C07284=1060.234,-74.990,436.185,171.327,26.753,155.011
C07285=1060.227,-75.240,436.197,171.325,26.751,155.011
C07286=1060.222,-75.490,436.207,171.323,26.750,155.011
C07287=1060.215,-75.739,436.219,171.321,26.748,155.011
C07288=1060.208,-75.989,436.230,171.319,26.747,155.011
C07289=1060.202,-76.239,436.241,171.318,26.745,155.011
C07290=1060.196,-76.488,436.252,171.316,26.744,155.011
C07291=1060.190,-76.738,436.263,171.314,26.743,155.011
C07292=1060.184,-76.987,436.275,171.312,26.741,155.011
C07293=1060.178,-77.238,436.286,171.311,26.739,155.010
C07294=1060.172,-77.487,436.297,171.309,26.738,155.010
C07295=1060.166,-77.737,436.308,171.307,26.736,155.010
C07296=1060.159,-77.986,436.320,171.306,26.735,155.010
C07297=1060.154,-78.236,436.330,171.304,26.733,155.010
C07298=1060.147,-78.486,436.342,171.302,26.732,155.010
C07299=1060.142,-78.735,436.353,171.301,26.731,155.010
C07300=1060.135,-78.985,436.364,171.299,26.729,155.010
C07301=1060.130,-79.235,436.375,171.297,26.728,155.010
C07302=1060.123,-79.485,436.387,171.294,26.726,155.010
C07303=1060.117,-79.734,436.398,171.293,26.725,155.010
C07304=1060.111,-79.983,436.408,171.291,26.723,155.010
C07305=1060.104,-80.233,436.419,171.289,26.722,155.010
C07306=1060.099,-80.483,436.430,171.288,26.721,155.010
C07307=1060.092,-80.733,436.441,171.286,26.719,155.009
C07308=1060.086,-80.982,436.451,171.284,26.718,155.009
C07309=1060.079,-81.232,436.463,171.282,26.716,155.009
C07310=1060.074,-81.482,436.474,171.281,26.715,155.009
C07311=1060.067,-81.732,436.485,171.279,26.714,155.009
C07312=1060.061,-81.981,436.495,171.277,26.712,155.009
C07313=1060.054,-82.264,436.508,171.275,26.711,155.009
C07314=1060.047,-82.546,436.520,171.273,26.709,155.009
C07315=1060.039,-82.829,436.533,171.271,26.708,155.009
C07316=1060.033,-83.111,436.545,171.269,26.706,155.009
C07317=1060.026,-83.361,436.555,171.267,26.704,155.009
C07318=1060.021,-83.611,436.566,171.265,26.703,155.009
C07319=1060.014,-83.861,436.578,171.263,26.702,155.009
C07320=1060.008,-84.110,436.588,171.262,26.700,155.009
C07321=1060.002,-84.359,436.599,171.260,26.699,155.009
C07322=1059.996,-84.610,436.610,171.258,26.698,155.008
C07323=1059.990,-84.859,436.621,171.256,26.696,155.008
C07324=1059.983,-85.109,436.632,171.255,26.695,155.008
C07325=1059.977,-85.359,436.642,171.253,26.694,155.008
C07326=1059.971,-85.608,436.653,171.251,26.692,155.008
C07327=1059.964,-85.858,436.664,171.249,26.691,155.008
C07328=1059.959,-86.107,436.675,171.248,26.690,155.008
C07329=1059.953,-86.357,436.686,171.245,26.688,155.008
C07330=1059.946,-86.607,436.696,171.243,26.687,155.008
C07331=1059.940,-86.856,436.707,171.242,26.686,155.008
C07332=1059.934,-87.106,436.718,171.240,26.684,155.008
C07333=1059.927,-87.356,436.729,171.238,26.683,155.008
C07334=1059.921,-87.605,436.740,171.236,26.682,155.008
C07335=1059.915,-87.855,436.751,171.235,26.681,155.008
C07336=1059.909,-88.105,436.760,171.233,26.679,155.008
C07337=1059.903,-88.355,436.771,171.231,26.678,155.008
C07338=1059.897,-88.604,436.782,171.229,26.677,155.008
C07339=1059.890,-88.854,436.793,171.228,26.676,155.008
C07340=1059.885,-89.103,436.804,171.226,26.674,155.007
C07341=1059.879,-89.353,436.815,171.224,26.673,155.007
C07342=1059.872,-89.603,436.824,171.222,26.672,155.007
C07343=1059.866,-89.853,436.835,171.220,26.670,155.007
C07344=1059.861,-90.102,436.846,171.218,26.669,155.007
C07345=1059.854,-90.352,436.857,171.216,26.667,155.007
C07346=1059.848,-90.602,436.868,171.215,26.666,155.007
C07347=1059.841,-90.851,436.878,171.213,26.665,155.007
C07348=1059.836,-91.101,436.888,171.211,26.664,155.007
C07349=1059.830,-91.351,436.899,171.209,26.663,155.007
C07350=1059.823,-91.600,436.910,171.208,26.662,155.007
C07351=1059.817,-91.850,436.921,171.206,26.660,155.007
C07352=1059.812,-92.100,436.931,171.204,26.659,155.007
C07353=1059.805,-92.350,436.941,171.202,26.658,155.007
C07354=1059.799,-92.599,436.952,171.201,26.656,155.007
C07355=1059.793,-92.849,436.963,171.199,26.655,155.007
C07356=1059.787,-93.099,436.973,171.197,26.654,155.007
C07357=1059.781,-93.349,436.984,171.194,26.653,155.007
C07358=1059.774,-93.598,436.994,171.193,26.651,155.007
C07359=1059.769,-93.848,437.004,171.191,26.650,155.007
C07360=1059.762,-94.097,437.015,171.189,26.649,155.007
C07361=1059.757,-94.347,437.026,171.187,26.648,155.007
C07362=1059.750,-94.597,437.037,171.186,26.646,155.007
C07363=1059.744,-94.847,437.046,171.184,26.645,155.007
C07364=1059.738,-95.096,437.057,171.182,26.644,155.007
C07365=1059.732,-95.346,437.067,171.180,26.643,155.007
C07366=1059.727,-95.596,437.078,171.179,26.642,155.007
C07367=1059.719,-95.846,437.088,171.177,26.641,155.007
C07368=1059.714,-96.096,437.099,171.175,26.639,155.006
C07369=1059.708,-96.345,437.109,171.173,26.638,155.006
C07370=1059.702,-96.594,437.120,171.172,26.637,155.006
C07371=1059.696,-96.844,437.130,171.169,26.635,155.006
C07372=1059.690,-97.094,437.140,171.167,26.634,155.006
C07373=1059.684,-97.344,437.150,171.165,26.633,155.006
C07374=1059.677,-97.594,437.161,171.164,26.632,155.006
C07375=1059.672,-97.843,437.172,171.162,26.631,155.006
C07376=1059.666,-98.093,437.181,171.160,26.629,155.006
C07377=1059.659,-98.377,437.193,171.158,26.628,155.006
C07378=1059.651,-98.662,437.205,171.156,26.627,155.006
C07379=1059.644,-98.947,437.217,171.154,26.626,155.006
C07380=1059.637,-99.232,437.229,171.152,26.625,155.006
C07381=1059.631,-99.482,437.238,171.150,26.623,155.006
C07382=1059.625,-99.731,437.249,171.148,26.623,155.006
C07383=1059.619,-99.981,437.259,171.146,26.622,155.006
C07384=1059.612,-100.231,437.270,171.144,26.620,155.006
C07385=1059.606,-100.481,437.279,171.142,26.619,155.006
C07386=1059.600,-100.730,437.290,171.140,26.618,155.006
C07387=1059.594,-100.980,437.300,171.139,26.617,155.006
C07388=1059.588,-101.230,437.309,171.137,26.616,155.006
C07389=1059.582,-101.479,437.320,171.135,26.615,155.006
C07390=1059.576,-101.729,437.330,171.133,26.614,155.006
C07391=1059.569,-101.979,437.340,171.132,26.613,155.006
C07392=1059.563,-102.229,437.350,171.130,26.612,155.006
C07393=1059.557,-102.478,437.361,171.128,26.611,155.006
C07394=1059.551,-102.728,437.370,171.126,26.610,155.006
C07395=1059.545,-102.977,437.381,171.123,26.609,155.006
C07396=1059.539,-103.227,437.391,171.122,26.608,155.006
C07397=1059.533,-103.477,437.400,171.120,26.606,155.006
C07398=1059.527,-103.726,437.411,171.118,26.606,155.007
C07399=1059.521,-103.976,437.421,171.116,26.605,155.006
C07400=1059.515,-104.226,437.430,171.114,26.604,155.006
C07401=1059.508,-104.476,437.442,171.113,26.602,155.006
C07402=1059.502,-104.726,437.451,171.111,26.602,155.007
C07403=1059.496,-104.975,437.461,171.109,26.601,155.007
C07404=1059.489,-105.225,437.471,171.107,26.600,155.007
C07405=1059.484,-105.475,437.481,171.106,26.598,155.006
C07406=1059.478,-105.724,437.491,171.104,26.598,155.007
C07407=1059.471,-105.974,437.501,171.102,26.597,155.007
C07408=1059.465,-106.224,437.511,171.099,26.595,155.007
C07409=1059.459,-106.473,437.521,171.097,26.595,155.007
C07410=1059.453,-106.723,437.531,171.096,26.594,155.007
C07411=1059.447,-106.973,437.541,171.094,26.592,155.007
C07412=1059.441,-107.223,437.550,171.092,26.592,155.007
C07413=1059.435,-107.472,437.561,171.090,26.591,155.007
C07414=1059.429,-107.722,437.571,171.088,26.590,155.007
C07415=1059.423,-107.972,437.580,171.087,26.589,155.007
C07416=1059.417,-108.222,437.590,171.085,26.588,155.007
C07417=1059.410,-108.472,437.600,171.083,26.587,155.007
C07418=1059.403,-108.721,437.610,171.081,26.586,155.007
C07419=1059.397,-108.971,437.619,171.079,26.585,155.007
C07420=1059.392,-109.221,437.630,171.077,26.584,155.007
C07421=1059.385,-109.470,437.640,171.075,26.583,155.007
C07422=1059.379,-109.720,437.649,171.073,26.583,155.007
C07423=1059.373,-109.970,437.659,171.071,26.581,155.007
C07424=1059.367,-110.220,437.669,171.069,26.581,155.007
C07425=1059.361,-110.470,437.678,171.068,26.580,155.007
C07426=1059.354,-110.719,437.688,171.066,26.579,155.007
C07427=1059.348,-110.969,437.698,171.064,26.578,155.007
C07428=1059.342,-111.218,437.708,171.062,26.577,155.007
C07429=1059.336,-111.469,437.718,171.060,26.576,155.007
C07430=1059.330,-111.718,437.727,171.058,26.576,155.007
C07431=1059.324,-111.968,437.737,171.057,26.575,155.007
C07432=1059.318,-112.218,437.746,171.055,26.574,155.007
C07433=1059.311,-112.467,437.757,171.053,26.573,155.007
C07434=1059.305,-112.717,437.766,171.050,26.572,155.008
C07435=1059.299,-112.967,437.776,171.048,26.571,155.008
C07436=1059.293,-113.217,437.785,171.047,26.570,155.008
C07437=1059.287,-113.466,437.795,171.045,26.569,155.008
C07438=1059.281,-113.716,437.805,171.043,26.569,155.008
C07439=1059.275,-113.965,437.814,171.041,26.567,155.008
C07440=1059.269,-114.215,437.823,171.039,26.567,155.008
C07441=1059.262,-114.499,437.834,171.037,26.566,155.008
C07442=1059.255,-114.782,437.846,171.035,26.565,155.008
C07443=1059.248,-115.065,437.857,171.033,26.564,155.008
C07444=1059.241,-115.348,437.867,171.031,26.563,155.008
C07445=1059.235,-115.598,437.877,171.029,26.563,155.008
C07446=1059.229,-115.847,437.886,171.026,26.561,155.008
C07447=1059.222,-116.097,437.896,171.025,26.561,155.008
C07448=1059.216,-116.347,437.905,171.023,26.560,155.008
C07449=1059.210,-116.597,437.915,171.021,26.559,155.008
C07450=1059.204,-116.847,437.924,171.019,26.558,155.008
C07451=1059.198,-117.096,437.934,171.017,26.558,155.009
C07452=1059.192,-117.346,437.944,171.015,26.557,155.008
C07453=1059.185,-117.596,437.953,171.014,26.556,155.009
C07454=1059.179,-117.846,437.963,171.012,26.556,155.009
C07455=1059.174,-118.095,437.972,171.010,26.555,155.009
C07456=1059.167,-118.345,437.981,171.008,26.554,155.009
C07457=1059.161,-118.594,437.991,171.006,26.553,155.009
C07458=1059.155,-118.844,438.001,171.004,26.553,155.009
C07459=1059.148,-119.094,438.010,171.001,26.552,155.009
C07460=1059.142,-119.344,438.019,171.000,26.551,155.009
C07461=1059.136,-119.593,438.029,170.998,26.550,155.009
C07462=1059.130,-119.844,438.038,170.996,26.550,155.009
C07463=1059.124,-120.094,438.047,170.994,26.549,155.009
C07464=1059.118,-120.343,438.056,170.992,26.548,155.009
C07465=1059.112,-120.592,438.066,170.990,26.547,155.009
C07466=1059.106,-120.842,438.075,170.989,26.547,155.010
C07467=1059.100,-121.092,438.085,170.987,26.546,155.010
C07468=1059.093,-121.342,438.094,170.985,26.546,155.010
C07469=1059.087,-121.592,438.103,170.983,26.545,155.010
C07470=1059.081,-121.842,438.112,170.981,26.544,155.010
C07471=1059.075,-122.091,438.122,170.979,26.544,155.010
C07472=1059.069,-122.341,438.131,170.976,26.543,155.010
C07473=1059.063,-122.590,438.141,170.975,26.542,155.010
C07474=1059.057,-122.840,438.150,170.973,26.542,155.010
C07475=1059.050,-123.090,438.159,170.971,26.541,155.010
C07476=1059.044,-123.340,438.168,170.969,26.540,155.010
C07477=1059.038,-123.589,438.177,170.967,26.539,155.010
C07478=1059.032,-123.839,438.187,170.965,26.539,155.011
C07479=1059.026,-124.089,438.196,170.963,26.538,155.011
C07480=1059.020,-124.339,438.205,170.962,26.538,155.011
C07481=1059.013,-124.589,438.214,170.960,26.537,155.011
C07482=1059.008,-124.838,438.223,170.958,26.537,155.011
C07483=1059.002,-125.088,438.232,170.956,26.536,155.011
C07484=1058.996,-125.338,438.242,170.954,26.536,155.011
C07485=1058.989,-125.588,438.251,170.952,26.535,155.011
C07486=1058.983,-125.837,438.260,170.949,26.534,155.011
C07487=1058.977,-126.088,438.269,170.948,26.534,155.011
C07488=1058.970,-126.337,438.278,170.946,26.533,155.012
C07489=1058.964,-126.586,438.287,170.944,26.532,155.012
C07490=1058.958,-126.837,438.296,170.942,26.532,155.012
C07491=1058.952,-127.087,438.306,170.940,26.531,155.012
C07492=1058.946,-127.335,438.314,170.938,26.531,155.012
C07493=1058.940,-127.586,438.323,170.936,26.530,155.012
C07494=1058.934,-127.836,438.333,170.934,26.530,155.012
C07495=1058.929,-128.085,438.343,170.933,26.529,155.012
C07496=1058.925,-128.335,438.352,170.931,26.527,155.012
C07497=1058.923,-128.586,438.364,170.929,26.525,155.012
C07498=1058.921,-128.837,438.375,170.928,26.522,155.012
C07499=1058.922,-129.087,438.388,170.927,26.519,155.011
C07500=1058.923,-129.337,438.401,170.926,26.515,155.011
C07501=1058.926,-129.589,438.415,170.925,26.511,155.010
C07502=1058.931,-129.840,438.429,170.924,26.505,155.009
C07503=1058.937,-130.091,438.445,170.924,26.500,155.008
C07504=1058.944,-130.341,438.461,170.923,26.494,155.007
C07505=1058.567,-130.364,438.262,170.876,26.654,155.040
C07506=1058.559,-130.114,438.246,170.876,26.661,155.041
C07507=1058.554,-129.864,438.232,170.877,26.666,155.042
C07508=1058.550,-129.612,438.217,170.878,26.671,155.043
C07509=1058.547,-129.361,438.203,170.878,26.676,155.044
C07510=1058.544,-129.110,438.189,170.879,26.680,155.044
C07511=1058.545,-128.860,438.177,170.880,26.683,155.045
C07512=1058.545,-128.609,438.165,170.882,26.686,155.045
C07513=1058.547,-128.358,438.154,170.883,26.688,155.045
C07514=1058.551,-128.109,438.144,170.884,26.690,155.045
C07515=1058.556,-127.859,438.135,170.886,26.691,155.046
C07516=1058.562,-127.609,438.125,170.889,26.692,155.045
C07517=1058.568,-127.359,438.115,170.891,26.692,155.045
C07518=1058.574,-127.109,438.107,170.893,26.692,155.045
C07519=1058.581,-126.860,438.098,170.894,26.693,155.045
C07520=1058.587,-126.610,438.088,170.896,26.693,155.045
C07521=1058.593,-126.360,438.080,170.898,26.694,155.045
C07522=1058.599,-126.110,438.071,170.900,26.694,155.045
C07523=1058.606,-125.860,438.061,170.902,26.695,155.045
C07524=1058.611,-125.611,438.052,170.904,26.695,155.044
C07525=1058.617,-125.361,438.043,170.906,26.696,155.044
C07526=1058.624,-125.111,438.034,170.908,26.696,155.044
C07527=1058.630,-124.861,438.024,170.910,26.697,155.044
C07528=1058.636,-124.611,438.016,170.912,26.698,155.044
C07529=1058.642,-124.361,438.006,170.914,26.698,155.044
C07530=1058.648,-124.112,437.997,170.916,26.699,155.044
C07531=1058.655,-123.863,437.988,170.918,26.700,155.044
C07532=1058.661,-123.613,437.978,170.920,26.701,155.044
C07533=1058.667,-123.362,437.969,170.922,26.701,155.044
C07534=1058.673,-123.113,437.960,170.924,26.702,155.044
C07535=1058.678,-122.864,437.951,170.925,26.702,155.043
C07536=1058.685,-122.614,437.942,170.927,26.703,155.043
C07537=1058.691,-122.364,437.933,170.929,26.703,155.043
C07538=1058.697,-122.114,437.923,170.931,26.704,155.043
C07539=1058.704,-121.864,437.914,170.933,26.705,155.043
C07540=1058.710,-121.614,437.904,170.935,26.705,155.043
C07541=1058.715,-121.365,437.895,170.937,26.706,155.043
C07542=1058.721,-121.115,437.885,170.939,26.707,155.043
C07543=1058.728,-120.866,437.876,170.941,26.707,155.043
C07544=1058.734,-120.615,437.868,170.943,26.708,155.043
C07545=1058.740,-120.366,437.858,170.945,26.709,155.043
C07546=1058.747,-120.116,437.848,170.947,26.710,155.043
C07547=1058.753,-119.866,437.839,170.949,26.710,155.042
C07548=1058.759,-119.616,437.829,170.951,26.711,155.042
C07549=1058.764,-119.367,437.820,170.952,26.712,155.042
C07550=1058.771,-119.117,437.811,170.954,26.712,155.042
C07551=1058.777,-118.868,437.801,170.956,26.713,155.042
C07552=1058.783,-118.618,437.791,170.958,26.713,155.042
C07553=1058.790,-118.368,437.782,170.961,26.715,155.042
C07554=1058.796,-118.118,437.774,170.963,26.715,155.042
C07555=1058.802,-117.868,437.764,170.964,26.716,155.042
C07556=1058.808,-117.618,437.754,170.966,26.716,155.042
C07557=1058.814,-117.368,437.745,170.968,26.718,155.042
C07558=1058.820,-117.119,437.735,170.970,26.718,155.042
C07559=1058.826,-116.870,437.726,170.972,26.719,155.042
C07560=1058.832,-116.620,437.717,170.974,26.720,155.042
C07561=1058.838,-116.370,437.707,170.975,26.720,155.042
C07562=1058.845,-116.120,437.697,170.977,26.721,155.041
C07563=1058.851,-115.870,437.688,170.979,26.722,155.041
C07564=1058.857,-115.621,437.678,170.981,26.723,155.041
C07565=1058.863,-115.371,437.669,170.984,26.723,155.041
C07566=1058.870,-115.087,437.658,170.986,26.725,155.041
C07567=1058.878,-114.804,437.647,170.987,26.725,155.041
C07568=1058.884,-114.522,437.636,170.990,26.726,155.041
C07569=1058.891,-114.238,437.625,170.992,26.727,155.041
C07570=1058.897,-113.988,437.615,170.994,26.728,155.041
C07571=1058.903,-113.738,437.606,170.996,26.729,155.041
C07572=1058.910,-113.489,437.596,170.998,26.729,155.041
C07573=1058.916,-113.239,437.587,170.999,26.730,155.041
C07574=1058.922,-112.989,437.577,171.001,26.731,155.041
C07575=1058.928,-112.740,437.567,171.003,26.732,155.041
C07576=1058.934,-112.490,437.557,171.006,26.733,155.041
C07577=1058.941,-112.240,437.548,171.008,26.734,155.041
C07578=1058.946,-111.990,437.538,171.009,26.735,155.041
C07579=1058.952,-111.740,437.528,171.011,26.735,155.040
C07580=1058.958,-111.490,437.519,171.013,26.736,155.041
C07581=1058.965,-111.241,437.509,171.015,26.737,155.040
C07582=1058.971,-110.992,437.499,171.017,26.738,155.040
C07583=1058.977,-110.742,437.489,171.019,26.739,155.040
C07584=1058.983,-110.492,437.480,171.020,26.740,155.040
C07585=1058.990,-110.242,437.470,171.022,26.741,155.040
C07586=1058.996,-109.992,437.460,171.024,26.741,155.040
C07587=1059.002,-109.743,437.451,171.026,26.743,155.040
C07588=1059.008,-109.493,437.440,171.029,26.743,155.040
C07589=1059.014,-109.243,437.430,171.030,26.744,155.040
C07590=1059.020,-108.993,437.421,171.032,26.745,155.040
C07591=1059.026,-108.744,437.411,171.034,26.746,155.040
C07592=1059.033,-108.494,437.401,171.036,26.747,155.040
C07593=1059.039,-108.245,437.391,171.038,26.748,155.040
C07594=1059.045,-107.995,437.382,171.040,26.748,155.040
C07595=1059.051,-107.745,437.372,171.041,26.750,155.040
C07596=1059.057,-107.496,437.361,171.043,26.751,155.040
C07597=1059.063,-107.246,437.352,171.045,26.751,155.040
C07598=1059.069,-106.996,437.342,171.047,26.752,155.040
C07599=1059.075,-106.746,437.333,171.049,26.753,155.040
C07600=1059.082,-106.496,437.321,171.051,26.754,155.040
C07601=1059.088,-106.246,437.312,171.053,26.755,155.040
C07602=1059.094,-105.996,437.302,171.055,26.757,155.040
C07603=1059.101,-105.747,437.292,171.057,26.757,155.040
C07604=1059.106,-105.497,437.282,171.059,26.758,155.040
C07605=1059.112,-105.247,437.272,171.060,26.759,155.040
C07606=1059.119,-104.998,437.262,171.062,26.760,155.040
C07607=1059.125,-104.748,437.252,171.064,26.761,155.040
C07608=1059.130,-104.498,437.242,171.066,26.762,155.040
C07609=1059.137,-104.249,437.232,171.067,26.763,155.040
C07610=1059.143,-103.999,437.222,171.069,26.764,155.040
C07611=1059.148,-103.749,437.212,171.071,26.765,155.040
C07612=1059.155,-103.500,437.202,171.073,26.766,155.040
C07613=1059.162,-103.249,437.192,171.076,26.768,155.040
C07614=1059.168,-103.000,437.182,171.077,26.768,155.040
C07615=1059.174,-102.750,437.172,171.079,26.769,155.040
C07616=1059.180,-102.501,437.161,171.081,26.770,155.040
C07617=1059.186,-102.251,437.152,171.083,26.772,155.040
C07618=1059.192,-102.001,437.142,171.085,26.773,155.040
C07619=1059.198,-101.752,437.131,171.086,26.773,155.040
C07620=1059.204,-101.502,437.122,171.088,26.774,155.040
C07621=1059.210,-101.253,437.111,171.090,26.775,155.040
C07622=1059.217,-101.002,437.101,171.092,26.777,155.040
C07623=1059.223,-100.753,437.091,171.094,26.778,155.040
C07624=1059.229,-100.503,437.080,171.095,26.778,155.040
C07625=1059.235,-100.254,437.070,171.098,26.780,155.040
C07626=1059.241,-100.004,437.061,171.100,26.781,155.040
C07627=1059.247,-99.754,437.050,171.102,26.782,155.040
C07628=1059.254,-99.504,437.040,171.103,26.783,155.040
C07629=1059.260,-99.254,437.029,171.105,26.784,155.040
C07630=1059.267,-98.969,437.018,171.107,26.785,155.040
C07631=1059.273,-98.685,437.006,171.110,26.787,155.040
C07632=1059.281,-98.399,436.994,171.111,26.788,155.040
C07633=1059.288,-98.115,436.983,171.113,26.789,155.040
C07634=1059.294,-97.865,436.973,171.115,26.790,155.040
C07635=1059.300,-97.616,436.962,171.118,26.792,155.040
C07636=1059.307,-97.367,436.952,171.120,26.792,155.040
C07637=1059.313,-97.116,436.942,171.121,26.793,155.040
C07638=1059.318,-96.866,436.931,171.123,26.795,155.040
C07639=1059.325,-96.617,436.921,171.125,26.796,155.040
C07640=1059.330,-96.367,436.910,171.127,26.797,155.040
C07641=1059.337,-96.118,436.900,171.128,26.798,155.040
C07642=1059.342,-95.868,436.890,171.130,26.800,155.040
C07643=1059.349,-95.618,436.879,171.132,26.801,155.040
C07644=1059.355,-95.368,436.868,171.134,26.802,155.040
C07645=1059.361,-95.118,436.858,171.135,26.803,155.040
C07646=1059.367,-94.869,436.848,171.137,26.804,155.040
C07647=1059.373,-94.620,436.837,171.139,26.805,155.040
C07648=1059.379,-94.370,436.827,171.142,26.807,155.040
C07649=1059.385,-94.120,436.816,171.143,26.808,155.040
C07650=1059.391,-93.870,436.805,171.145,26.809,155.040
C07651=1059.397,-93.620,436.796,171.147,26.811,155.040
C07652=1059.403,-93.371,436.785,171.149,26.812,155.040
C07653=1059.410,-93.121,436.774,171.150,26.813,155.040
C07654=1059.415,-92.871,436.764,171.152,26.814,155.040
C07655=1059.421,-92.621,436.753,171.154,26.815,155.040
C07656=1059.428,-92.372,436.743,171.156,26.816,155.040
C07657=1059.433,-92.123,436.732,171.157,26.817,155.040
C07658=1059.440,-91.872,436.722,171.159,26.819,155.040
C07659=1059.446,-91.623,436.711,171.161,26.820,155.040
C07660=1059.452,-91.373,436.700,171.163,26.821,155.040
C07661=1059.459,-91.123,436.690,171.164,26.823,155.040
C07662=1059.464,-90.874,436.679,171.167,26.824,155.040
C07663=1059.470,-90.624,436.669,171.169,26.825,155.040
C07664=1059.476,-90.375,436.658,171.171,26.826,155.040
C07665=1059.483,-90.124,436.647,171.172,26.828,155.041
C07666=1059.489,-89.875,436.637,171.174,26.829,155.041
C07667=1059.495,-89.626,436.626,171.176,26.830,155.041
C07668=1059.501,-89.375,436.615,171.178,26.831,155.041
C07669=1059.507,-89.126,436.605,171.179,26.833,155.041
C07670=1059.513,-88.876,436.594,171.181,26.834,155.041
C07671=1059.519,-88.627,436.583,171.183,26.835,155.041
C07672=1059.526,-88.377,436.573,171.185,26.837,155.041
C07673=1059.532,-88.127,436.562,171.186,26.838,155.041
C07674=1059.537,-87.878,436.551,171.188,26.839,155.041
C07675=1059.544,-87.627,436.541,171.191,26.841,155.041
C07676=1059.550,-87.378,436.530,171.193,26.842,155.041
C07677=1059.556,-87.128,436.519,171.194,26.843,155.041
C07678=1059.563,-86.879,436.509,171.196,26.845,155.041
C07679=1059.569,-86.629,436.498,171.198,26.846,155.041
C07680=1059.574,-86.380,436.487,171.200,26.847,155.041
C07681=1059.581,-86.130,436.476,171.201,26.848,155.041
C07682=1059.587,-85.880,436.465,171.203,26.850,155.041
C07683=1059.593,-85.630,436.454,171.205,26.851,155.041
C07684=1059.600,-85.381,436.444,171.207,26.852,155.041
C07685=1059.606,-85.131,436.433,171.208,26.853,155.041
C07686=1059.612,-84.881,436.422,171.210,26.855,155.042
C07687=1059.618,-84.632,436.411,171.212,26.856,155.042
C07688=1059.625,-84.382,436.400,171.213,26.857,155.042
C07689=1059.631,-84.132,436.389,171.216,26.859,155.042
C07690=1059.636,-83.883,436.378,171.218,26.860,155.042
C07691=1059.643,-83.633,436.368,171.220,26.862,155.042
C07692=1059.649,-83.383,436.357,171.221,26.863,155.042
C07693=1059.655,-83.133,436.346,171.223,26.864,155.042
C07694=1059.662,-82.851,436.334,171.225,26.866,155.042
C07695=1059.669,-82.569,436.322,171.227,26.868,155.042
C07696=1059.676,-82.286,436.309,171.229,26.869,155.042
C07697=1059.684,-82.004,436.296,171.231,26.870,155.042
C07698=1059.689,-81.754,436.286,171.233,26.872,155.042
C07699=1059.696,-81.504,436.274,171.234,26.873,155.042
C07700=1059.702,-81.255,436.264,171.236,26.874,155.042
C07701=1059.709,-81.004,436.253,171.239,26.876,155.042
C07702=1059.714,-80.755,436.242,171.240,26.878,155.043
C07703=1059.721,-80.505,436.231,171.242,26.879,155.043
C07704=1059.727,-80.256,436.220,171.244,26.880,155.043
C07705=1059.733,-80.005,436.209,171.246,26.882,155.043
C07706=1059.739,-79.756,436.198,171.247,26.883,155.043
C07707=1059.746,-79.506,436.187,171.249,26.884,155.043
C07708=1059.752,-79.257,436.175,171.251,26.885,155.043
C07709=1059.758,-79.007,436.164,171.253,26.887,155.043
C07710=1059.764,-78.758,436.154,171.254,26.888,155.043
C07711=1059.770,-78.508,436.143,171.256,26.890,155.043
C07712=1059.777,-78.258,436.132,171.258,26.892,155.043
C07713=1059.783,-78.009,436.120,171.259,26.893,155.043
C07714=1059.789,-77.759,436.109,171.261,26.895,155.044
C07715=1059.795,-77.509,436.098,171.263,26.896,155.044
C07716=1059.801,-77.259,436.087,171.265,26.898,155.044
C07717=1059.807,-77.010,436.076,171.267,26.899,155.044
C07718=1059.813,-76.760,436.064,171.269,26.901,155.044
C07719=1059.819,-76.511,436.053,171.271,26.902,155.044
C07720=1059.825,-76.260,436.042,171.272,26.903,155.044
C07721=1059.831,-76.011,436.031,171.274,26.905,155.044
C07722=1059.838,-75.761,436.019,171.276,26.906,155.044
C07723=1059.844,-75.512,436.008,171.277,26.908,155.044
C07724=1059.850,-75.262,435.997,171.279,26.909,155.044
C07725=1059.856,-75.012,435.986,171.281,26.911,155.044
C07726=1059.862,-74.763,435.974,171.283,26.913,155.045
C07727=1059.868,-74.513,435.963,171.284,26.914,155.045
C07728=1059.874,-74.263,435.952,171.286,26.915,155.045
C07729=1059.880,-74.014,435.940,171.288,26.917,155.045
C07730=1059.887,-73.764,435.929,171.289,26.918,155.045
C07731=1059.893,-73.514,435.918,171.291,26.920,155.045
C07732=1059.899,-73.265,435.906,171.293,26.922,155.045
C07733=1059.904,-73.015,435.895,171.295,26.924,155.045
C07734=1059.910,-72.765,435.884,171.297,26.925,155.045
C07735=1059.917,-72.516,435.872,171.299,26.927,155.045
C07736=1059.923,-72.266,435.861,171.301,26.928,155.046
C07737=1059.929,-72.016,435.850,171.302,26.930,155.046
C07738=1059.935,-71.766,435.837,171.304,26.932,155.046
C07739=1059.940,-71.517,435.826,171.306,26.933,155.046
C07740=1059.947,-71.267,435.814,171.307,26.935,155.046
C07741=1059.953,-71.018,435.804,171.309,26.936,155.046
C07742=1059.959,-70.768,435.792,171.311,26.938,155.046
C07743=1059.964,-70.518,435.780,171.312,26.940,155.046
C07744=1059.971,-70.268,435.769,171.314,26.941,155.047
C07745=1059.977,-70.019,435.757,171.316,26.943,155.047
C07746=1059.983,-69.769,435.746,171.317,26.944,155.047
C07747=1059.988,-69.520,435.734,171.319,26.946,155.047
C07748=1059.995,-69.270,435.723,171.321,26.948,155.047
C07749=1060.001,-69.020,435.711,171.322,26.949,155.047
C07750=1060.007,-68.771,435.700,171.324,26.951,155.047
C07751=1060.014,-68.521,435.688,171.326,26.953,155.047
C07752=1060.019,-68.271,435.676,171.328,26.954,155.048
C07753=1060.025,-68.022,435.664,171.330,26.956,155.048
C07754=1060.031,-67.772,435.654,171.332,26.958,155.048
C07755=1060.038,-67.523,435.642,171.333,26.959,155.048
C07756=1060.043,-67.272,435.630,171.335,26.961,155.048
C07757=1060.049,-67.023,435.618,171.337,26.963,155.048
C07758=1060.057,-66.742,435.605,171.338,26.965,155.048
C07759=1060.063,-66.462,435.592,171.340,26.966,155.048
C07760=1060.069,-66.182,435.579,171.343,26.968,155.049
C07761=1060.077,-65.902,435.566,171.344,26.970,155.049
C07762=1060.083,-65.653,435.554,171.346,26.972,155.049
C07763=1060.088,-65.402,435.542,171.348,26.973,155.049
C07764=1060.095,-65.153,435.530,171.349,26.975,155.049
C07765=1060.101,-64.903,435.520,171.351,26.977,155.049
C07766=1060.108,-64.654,435.508,171.353,26.979,155.049
C07767=1060.113,-64.404,435.495,171.354,26.980,155.050
C07768=1060.119,-64.154,435.484,171.356,26.982,155.050
C07769=1060.126,-63.905,435.472,171.358,26.984,155.050
C07770=1060.132,-63.655,435.460,171.359,26.985,155.050
C07771=1060.137,-63.405,435.449,171.361,26.987,155.050
C07772=1060.144,-63.156,435.437,171.363,26.989,155.050
C07773=1060.150,-62.906,435.424,171.364,26.991,155.050
C07774=1060.156,-62.656,435.413,171.367,26.993,155.051
C07775=1060.162,-62.407,435.401,171.369,26.994,155.051
C07776=1060.169,-62.157,435.389,171.371,26.995,155.051
C07777=1060.174,-61.907,435.378,171.372,26.997,155.051
C07778=1060.181,-61.658,435.366,171.374,26.999,155.051
C07779=1060.187,-61.408,435.354,171.376,27.001,155.051
C07780=1060.193,-61.158,435.342,171.377,27.002,155.051
C07781=1060.199,-60.909,435.331,171.379,27.004,155.051
C07782=1060.206,-60.659,435.319,171.381,27.006,155.052
C07783=1060.212,-60.409,435.306,171.382,27.007,155.052
C07784=1060.217,-60.160,435.295,171.384,27.009,155.052
C07785=1060.224,-59.910,435.283,171.386,27.011,155.052
C07786=1060.230,-59.660,435.271,171.387,27.013,155.052
C07787=1060.236,-59.411,435.259,171.389,27.014,155.052
C07788=1060.243,-59.162,435.247,171.391,27.016,155.052
C07789=1060.248,-58.912,435.235,171.392,27.018,155.053
C07790=1060.255,-58.662,435.223,171.394,27.019,155.053
C07791=1060.261,-58.412,435.211,171.395,27.022,155.053
C07792=1060.267,-58.163,435.199,171.397,27.023,155.053
C07793=1060.273,-57.914,435.187,171.399,27.025,155.053
C07794=1060.280,-57.663,435.176,171.401,27.027,155.053
C07795=1060.286,-57.414,435.164,171.402,27.029,155.054
C07796=1060.292,-57.164,435.152,171.404,27.030,155.054
C07797=1060.298,-56.915,435.139,171.406,27.032,155.054
C07798=1060.304,-56.665,435.127,171.407,27.034,155.054
C07799=1060.311,-56.416,435.115,171.410,27.036,155.054
C07800=1060.317,-56.166,435.103,171.411,27.037,155.054
C07801=1060.323,-55.916,435.092,171.413,27.039,155.054
C07802=1060.329,-55.667,435.080,171.415,27.041,155.055
C07803=1060.335,-55.417,435.068,171.417,27.043,155.055
C07804=1060.342,-55.167,435.056,171.418,27.044,155.055
C07805=1060.348,-54.917,435.043,171.420,27.046,155.055
C07806=1060.354,-54.668,435.031,171.422,27.048,155.055
C07807=1060.361,-54.418,435.019,171.423,27.050,155.055
C07808=1060.366,-54.169,435.007,171.425,27.052,155.055
C07809=1060.373,-53.919,434.995,171.426,27.053,155.056
C07810=1060.379,-53.670,434.982,171.428,27.055,155.056
C07811=1060.385,-53.420,434.970,171.430,27.057,155.056
C07812=1060.392,-53.170,434.958,171.431,27.059,155.056
C07813=1060.398,-52.921,434.946,171.433,27.060,155.056
C07814=1060.405,-52.671,434.934,171.435,27.062,155.056
C07815=1060.411,-52.421,434.921,171.436,27.064,155.057
C07816=1060.417,-52.172,434.910,171.438,27.066,155.057
C07817=1060.423,-51.923,434.898,171.440,27.068,155.057
C07818=1060.429,-51.673,434.885,171.441,27.069,155.057
C07819=1060.436,-51.423,434.873,171.443,27.071,155.057
C07820=1060.442,-51.173,434.861,171.445,27.073,155.057
C07821=1060.448,-50.924,434.849,171.446,27.074,155.057
C07822=1060.456,-50.645,434.835,171.448,27.077,155.058
C07823=1060.462,-50.365,434.822,171.451,27.079,155.058
C07824=1060.468,-50.086,434.808,171.452,27.081,155.058
C07825=1060.476,-49.807,434.794,171.454,27.083,155.058
C07826=1060.481,-49.557,434.781,171.455,27.085,155.059
C07827=1060.488,-49.308,434.770,171.457,27.087,155.059
C07828=1060.494,-49.058,434.757,171.459,27.088,155.059
C07829=1060.500,-48.809,434.744,171.460,27.091,155.059
C07830=1060.506,-48.560,434.732,171.462,27.092,155.059
C07831=1060.512,-48.310,434.720,171.464,27.094,155.059
C07832=1060.518,-48.060,434.707,171.465,27.096,155.060
C07833=1060.524,-47.810,434.694,171.467,27.098,155.060
C07834=1060.531,-47.561,434.682,171.469,27.100,155.060
C07835=1060.537,-47.311,434.670,171.470,27.102,155.060
C07836=1060.543,-47.061,434.657,171.472,27.104,155.060
C07837=1060.548,-46.812,434.644,171.473,27.106,155.061
C07838=1060.555,-46.563,434.633,171.475,27.108,155.061
C07839=1060.561,-46.313,434.620,171.477,27.110,155.061
C07840=1060.567,-46.063,434.607,171.478,27.112,155.061
C07841=1060.573,-45.814,434.594,171.481,27.114,155.061
C07842=1060.579,-45.564,434.582,171.483,27.116,155.062
C07843=1060.585,-45.314,434.570,171.484,27.118,155.062
C07844=1060.591,-45.064,434.557,171.486,27.120,155.062
C07845=1060.597,-44.815,434.544,171.488,27.122,155.062
C07846=1060.604,-44.566,434.532,171.489,27.124,155.062
C07847=1060.610,-44.316,434.519,171.491,27.126,155.062
C07848=1060.616,-44.066,434.507,171.492,27.128,155.063
C07849=1060.622,-43.816,434.493,171.494,27.130,155.063
C07850=1060.629,-43.567,434.482,171.496,27.132,155.063
C07851=1060.635,-43.317,434.469,171.497,27.133,155.063
C07852=1060.640,-43.068,434.456,171.499,27.136,155.063
C07853=1060.646,-42.819,434.443,171.501,27.137,155.064
C07854=1060.653,-42.569,434.432,171.502,27.140,155.064
C07855=1060.659,-42.319,434.419,171.504,27.141,155.064
C07856=1060.665,-42.070,434.406,171.505,27.144,155.064
C07857=1060.671,-41.820,434.393,171.507,27.145,155.064
C07858=1060.677,-41.570,434.381,171.509,27.148,155.065
C07859=1060.684,-41.321,434.368,171.510,27.149,155.065
C07860=1060.690,-41.071,434.355,171.512,27.151,155.065
C07861=1060.696,-40.822,434.342,171.514,27.153,155.065
C07862=1060.702,-40.572,434.330,171.515,27.155,155.065
C07863=1060.708,-40.322,434.317,171.517,27.157,155.066
C07864=1060.715,-40.073,434.304,171.519,27.159,155.066
C07865=1060.720,-39.823,434.292,171.520,27.161,155.066
C07866=1060.727,-39.573,434.279,171.522,27.163,155.066
C07867=1060.733,-39.324,434.266,171.523,27.165,155.066
C07868=1060.739,-39.074,434.253,171.525,27.167,155.067
C07869=1060.745,-38.824,434.240,171.527,27.169,155.067
C07870=1060.752,-38.575,434.228,171.528,27.171,155.067
C07871=1060.758,-38.326,434.215,171.530,27.173,155.067
C07872=1060.764,-38.076,434.202,171.532,27.175,155.067
C07873=1060.770,-37.826,434.189,171.533,27.177,155.068
C07874=1060.776,-37.577,434.176,171.535,27.180,155.068
C07875=1060.782,-37.327,434.163,171.536,27.181,155.068
C07876=1060.788,-37.077,434.150,171.538,27.184,155.068
C07877=1060.795,-36.828,434.137,171.540,27.186,155.069
C07878=1060.800,-36.578,434.124,171.541,27.187,155.069
C07879=1060.806,-36.329,434.111,171.543,27.190,155.069
C07880=1060.812,-36.079,434.098,171.544,27.192,155.069
C07881=1060.818,-35.830,434.085,171.546,27.194,155.069
C07882=1060.824,-35.580,434.072,171.548,27.196,155.070
C07883=1060.830,-35.330,434.059,171.549,27.198,155.070
C07884=1060.836,-35.080,434.046,171.551,27.200,155.070
C07885=1060.842,-34.831,434.033,171.553,27.202,155.070
C07886=1060.850,-34.552,434.019,171.554,27.205,155.071
C07887=1060.856,-34.273,434.004,171.556,27.207,155.071
C07888=1060.863,-33.996,433.990,171.557,27.209,155.071
C07889=1060.870,-33.716,433.976,171.559,27.211,155.071
C07890=1060.876,-33.467,433.962,171.561,27.213,155.072
C07891=1060.882,-33.218,433.949,171.562,27.215,155.072
C07892=1060.888,-32.968,433.937,171.564,27.218,155.072
C07893=1060.894,-32.719,433.923,171.565,27.219,155.072
C07894=1060.901,-32.469,433.910,171.567,27.222,155.073
C07895=1060.907,-32.219,433.897,171.569,27.224,155.073
C07896=1060.912,-31.969,433.883,171.570,27.226,155.073
C07897=1060.919,-31.720,433.870,171.572,27.228,155.073
C07898=1060.925,-31.470,433.857,171.573,27.230,155.073
C07899=1060.931,-31.221,433.844,171.575,27.232,155.074
C07900=1060.937,-30.972,433.831,171.577,27.234,155.074
C07901=1060.943,-30.722,433.818,171.578,27.237,155.074
C07902=1060.950,-30.472,433.805,171.580,27.239,155.074
C07903=1060.956,-30.222,433.791,171.581,27.241,155.075
C07904=1060.962,-29.973,433.779,171.583,27.243,155.075
C07905=1060.968,-29.723,433.766,171.585,27.245,155.075
C07906=1060.974,-29.474,433.752,171.586,27.247,155.075
C07907=1060.980,-29.225,433.739,171.588,27.249,155.076
C07908=1060.986,-28.974,433.726,171.589,27.251,155.076
C07909=1060.992,-28.725,433.712,171.591,27.254,155.076
C07910=1060.999,-28.475,433.699,171.593,27.255,155.076
C07911=1061.005,-28.226,433.686,171.594,27.258,155.076
C07912=1061.011,-27.976,433.673,171.596,27.260,155.077
C07913=1061.018,-27.726,433.660,171.598,27.262,155.077
C07914=1061.024,-27.477,433.646,171.599,27.264,155.077
C07915=1061.030,-27.228,433.633,171.601,27.266,155.077
C07916=1061.036,-26.978,433.620,171.602,27.268,155.078
C07917=1061.041,-26.728,433.607,171.604,27.270,155.078
C07918=1061.048,-26.478,433.593,171.606,27.272,155.078
C07919=1061.054,-26.229,433.580,171.607,27.275,155.078
C07920=1061.060,-25.979,433.566,171.609,27.277,155.079
C07921=1061.066,-25.730,433.553,171.610,27.279,155.079
C07922=1061.072,-25.481,433.539,171.612,27.282,155.079
C07923=1061.078,-25.231,433.525,171.614,27.284,155.079
C07924=1061.084,-24.981,433.512,171.615,27.286,155.080
C07925=1061.091,-24.731,433.499,171.617,27.288,155.080
C07926=1061.097,-24.482,433.486,171.618,27.290,155.080
C07927=1061.102,-24.233,433.472,171.619,27.292,155.080
C07928=1061.108,-23.983,433.459,171.621,27.294,155.081
C07929=1061.115,-23.733,433.445,171.622,27.297,155.081
C07930=1061.121,-23.484,433.431,171.624,27.299,155.081
C07931=1061.127,-23.235,433.418,171.625,27.301,155.081
C07932=1061.133,-22.985,433.405,171.627,27.304,155.082
C07933=1061.139,-22.736,433.391,171.629,27.306,155.082
C07934=1061.145,-22.486,433.377,171.630,27.307,155.082
C07935=1061.151,-22.236,433.363,171.632,27.310,155.082
C07936=1061.157,-21.987,433.350,171.633,27.312,155.083
C07937=1061.163,-21.738,433.337,171.635,27.314,155.083
C07938=1061.169,-21.487,433.323,171.637,27.317,155.083
C07939=1061.176,-21.238,433.309,171.638,27.319,155.083
C07940=1061.182,-20.989,433.296,171.640,27.321,155.084
C07941=1061.187,-20.739,433.282,171.641,27.323,155.084
C07942=1061.194,-20.489,433.269,171.643,27.326,155.084
C07943=1061.200,-20.240,433.255,171.645,27.328,155.085
C07944=1061.206,-19.991,433.241,171.646,27.330,155.085
C07945=1061.213,-19.741,433.228,171.648,27.332,155.085
C07946=1061.218,-19.491,433.214,171.649,27.334,155.085
C07947=1061.224,-19.242,433.201,171.651,27.337,155.085
C07948=1061.231,-18.992,433.187,171.653,27.339,155.086
C07949=1061.237,-18.742,433.173,171.654,27.341,155.086
C07950=1061.243,-18.463,433.158,171.656,27.343,155.086
C07951=1061.250,-18.183,433.143,171.657,27.346,155.087
C07952=1061.258,-17.904,433.128,171.659,27.348,155.087
C07953=1061.264,-17.625,433.112,171.660,27.351,155.087
C07954=1061.271,-17.375,433.098,171.662,27.353,155.087
C07955=1061.276,-17.125,433.085,171.664,27.355,155.088
C07956=1061.282,-16.876,433.071,171.665,27.358,155.088
C07957=1061.289,-16.626,433.058,171.667,27.360,155.088
C07958=1061.295,-16.377,433.043,171.668,27.362,155.089
C07959=1061.301,-16.128,433.030,171.670,27.364,155.089
C07960=1061.307,-15.878,433.016,171.672,27.367,155.089
C07961=1061.314,-15.628,433.002,171.673,27.369,155.089
C07962=1061.320,-15.378,432.989,171.675,27.371,155.090
C07963=1061.326,-15.129,432.975,171.676,27.373,155.090
C07964=1061.332,-14.880,432.961,171.678,27.376,155.090
C07965=1061.338,-14.630,432.947,171.680,27.378,155.090
C07966=1061.344,-14.380,432.933,171.681,27.380,155.091
C07967=1061.350,-14.131,432.919,171.683,27.383,155.091
C07968=1061.356,-13.881,432.905,171.683,27.385,155.091
C07969=1061.362,-13.632,432.891,171.685,27.387,155.092
C07970=1061.368,-13.382,432.877,171.687,27.389,155.092
C07971=1061.374,-13.132,432.863,171.688,27.391,155.092
C07972=1061.381,-12.884,432.849,171.690,27.394,155.092
C07973=1061.386,-12.634,432.835,171.691,27.397,155.093
C07974=1061.392,-12.384,432.821,171.693,27.399,155.093
C07975=1061.399,-12.134,432.808,171.694,27.401,155.093
C07976=1061.404,-11.886,432.793,171.696,27.403,155.093
C07977=1061.410,-11.635,432.779,171.698,27.406,155.094
C07978=1061.417,-11.386,432.766,171.699,27.408,155.094
C07979=1061.423,-11.136,432.751,171.701,27.410,155.094
C07980=1061.429,-10.887,432.738,171.702,27.412,155.095
C07981=1061.435,-10.637,432.724,171.704,27.415,155.095
C07982=1061.441,-10.388,432.709,171.705,27.418,155.095
C07983=1061.447,-10.139,432.695,171.707,27.420,155.095
C07984=1061.453,-9.888,432.681,171.708,27.422,155.096
C07985=1061.459,-9.639,432.667,171.709,27.424,155.096
C07986=1061.465,-9.390,432.653,171.711,27.426,155.096
C07987=1061.471,-9.140,432.639,171.713,27.429,155.097
C07988=1061.477,-8.891,432.625,171.714,27.431,155.097
C07989=1061.484,-8.641,432.611,171.716,27.433,155.097
C07990=1061.490,-8.392,432.596,171.717,27.435,155.097
C07991=1061.496,-8.142,432.582,171.719,27.438,155.098
C07992=1061.502,-7.892,432.569,171.720,27.441,155.098
C07993=1061.508,-7.643,432.554,171.722,27.443,155.098
C07994=1061.514,-7.393,432.540,171.724,27.445,155.099
C07995=1061.520,-7.144,432.526,171.725,27.447,155.099
C07996=1061.527,-6.894,432.512,171.727,27.450,155.099
C07997=1061.532,-6.645,432.497,171.728,27.452,155.099
C07998=1061.539,-6.395,432.484,171.729,27.454,155.100
C07999=1061.545,-6.146,432.469,171.731,27.457,155.100
C08000=1061.551,-5.896,432.455,171.732,27.459,155.100
C08001=1061.557,-5.647,432.440,171.734,27.461,155.101
C08002=1061.564,-5.397,432.427,171.735,27.464,155.101
C08003=1061.569,-5.148,432.412,171.737,27.466,155.101
C08004=1061.575,-4.898,432.398,171.739,27.468,155.101
C08005=1061.582,-4.649,432.384,171.740,27.470,155.102
C08006=1061.588,-4.399,432.370,171.742,27.473,155.102
C08007=1061.594,-4.150,432.355,171.743,27.476,155.102
C08008=1061.600,-3.900,432.341,171.745,27.478,155.103
C08009=1061.606,-3.651,432.327,171.746,27.480,155.103
C08010=1061.613,-3.401,432.313,171.748,27.482,155.103
C08011=1061.618,-3.152,432.298,171.749,27.484,155.103
C08012=1061.625,-2.902,432.283,171.750,27.487,155.104
C08013=1061.630,-2.653,432.269,171.752,27.489,155.104
C08014=1061.637,-2.372,432.253,171.753,27.492,155.105
C08015=1061.644,-2.091,432.236,171.756,27.495,155.105
C08016=1061.651,-1.810,432.221,171.757,27.498,155.105
C08017=1061.657,-1.529,432.204,171.759,27.500,155.106
C08018=1061.663,-1.279,432.189,171.760,27.503,155.106
C08019=1061.669,-1.030,432.175,171.762,27.506,155.106
C08020=1061.675,-0.780,432.160,171.764,27.508,155.106
C08021=1061.681,-0.530,432.146,171.765,27.510,155.107
C08022=1061.687,-0.281,432.131,171.766,27.513,155.107
C08023=1061.693,-0.032,432.116,171.767,27.515,155.107
C08024=1061.699,0.219,432.102,171.769,27.517,155.108
C08025=1061.705,0.468,432.087,171.770,27.520,155.108
C08026=1061.711,0.717,432.073,171.772,27.522,155.108
C08027=1061.717,0.967,432.058,171.774,27.525,155.109
C08028=1061.723,1.216,432.044,171.775,27.527,155.109
C08029=1061.729,1.466,432.029,171.777,27.530,155.109
C08030=1061.735,1.715,432.014,171.778,27.532,155.110
C08031=1061.741,1.965,432.000,171.780,27.534,155.110
C08032=1061.747,2.214,431.985,171.780,27.537,155.110
C08033=1061.753,2.464,431.971,171.782,27.539,155.111
C08034=1061.759,2.713,431.956,171.784,27.541,155.111
C08035=1061.765,2.963,431.942,171.785,27.544,155.111
C08036=1061.772,3.213,431.927,171.787,27.546,155.111
C08037=1061.777,3.462,431.912,171.788,27.549,155.112
C08038=1061.784,3.711,431.897,171.790,27.552,155.112
C08039=1061.790,3.960,431.883,171.792,27.554,155.112
C08040=1061.796,4.211,431.868,171.793,27.556,155.113
C08041=1061.801,4.460,431.854,171.795,27.559,155.113
C08042=1061.808,4.709,431.839,171.795,27.561,155.113
C08043=1061.814,4.959,431.824,171.797,27.563,155.114
C08044=1061.820,5.208,431.809,171.798,27.566,155.114
C08045=1061.826,5.457,431.794,171.800,27.568,155.114
C08046=1061.832,5.708,431.780,171.802,27.571,155.115
C08047=1061.838,5.957,431.766,171.803,27.573,155.115
C08048=1061.845,6.206,431.751,171.805,27.576,155.115
C08049=1061.850,6.455,431.736,171.806,27.579,155.116
C08050=1061.857,6.705,431.721,171.808,27.581,155.116
C08051=1061.863,6.955,431.706,171.809,27.583,155.116
C08052=1061.869,7.204,431.692,171.810,27.586,155.117
C08053=1061.875,7.453,431.677,171.812,27.588,155.117
C08054=1061.881,7.703,431.661,171.813,27.590,155.117
C08055=1061.887,7.952,431.647,171.815,27.593,155.117
C08056=1061.893,8.202,431.632,171.816,27.595,155.118
C08057=1061.899,8.452,431.617,171.818,27.597,155.118
C08058=1061.905,8.701,431.603,171.819,27.600,155.118
C08059=1061.911,8.951,431.588,171.821,27.603,155.119
C08060=1061.918,9.200,431.573,171.823,27.605,155.119
C08061=1061.924,9.449,431.558,171.824,27.608,155.119
C08062=1061.930,9.699,431.543,171.825,27.610,155.120
C08063=1061.936,9.949,431.528,171.826,27.612,155.120
C08064=1061.943,10.198,431.514,171.828,27.615,155.120
C08065=1061.948,10.447,431.499,171.830,27.617,155.121
C08066=1061.954,10.697,431.483,171.831,27.619,155.121
C08067=1061.961,10.947,431.468,171.833,27.622,155.121
C08068=1061.966,11.196,431.454,171.834,27.624,155.121
C08069=1061.973,11.446,431.439,171.836,27.627,155.122
C08070=1061.979,11.695,431.424,171.837,27.629,155.122
C08071=1061.985,11.945,431.409,171.838,27.631,155.122
C08072=1061.991,12.194,431.394,171.840,27.634,155.123
C08073=1061.998,12.443,431.380,171.841,27.637,155.123
C08074=1062.004,12.692,431.364,171.843,27.639,155.123
C08075=1062.010,12.942,431.348,171.844,27.642,155.124
C08076=1062.016,13.191,431.334,171.846,27.644,155.124
C08077=1062.022,13.441,431.319,171.848,27.646,155.124
C08078=1062.029,13.724,431.302,171.849,27.649,155.125
C08079=1062.037,14.007,431.285,171.851,27.652,155.125
C08080=1062.043,14.291,431.268,171.852,27.655,155.125
C08081=1062.051,14.573,431.251,171.854,27.657,155.126
C08082=1062.056,14.823,431.235,171.855,27.660,155.126
C08083=1062.062,15.072,431.221,171.857,27.663,155.127
C08084=1062.068,15.322,431.206,171.858,27.665,155.127
C08085=1062.074,15.571,431.190,171.860,27.668,155.127
C08086=1062.080,15.820,431.175,171.862,27.670,155.127
C08087=1062.087,16.070,431.160,171.863,27.672,155.128
C08088=1062.092,16.320,431.144,171.865,27.675,155.128
C08089=1062.098,16.569,431.130,171.865,27.677,155.128
C08090=1062.105,16.818,431.114,171.867,27.680,155.129
C08091=1062.110,17.068,431.098,171.868,27.682,155.129
C08092=1062.117,17.318,431.084,171.870,27.685,155.129
C08093=1062.123,17.567,431.069,171.872,27.687,155.130
C08094=1062.128,17.816,431.053,171.873,27.690,155.130
C08095=1062.135,18.065,431.038,171.875,27.692,155.130
C08096=1062.141,18.315,431.023,171.876,27.695,155.131
C08097=1062.147,18.565,431.007,171.877,27.697,155.131
C08098=1062.153,18.813,430.992,171.878,27.700,155.132
C08099=1062.159,19.063,430.977,171.880,27.702,155.132
C08100=1062.165,19.313,430.961,171.882,27.705,155.132
C08101=1062.172,19.562,430.946,171.883,27.707,155.132
C08102=1062.177,19.812,430.930,171.885,27.710,155.133
C08103=1062.184,20.062,430.915,171.886,27.712,155.133
C08104=1062.189,20.311,430.901,171.888,27.715,155.133
C08105=1062.195,20.560,430.884,171.889,27.717,155.134
C08106=1062.202,20.810,430.870,171.890,27.720,155.134
C08107=1062.207,21.060,430.854,171.892,27.722,155.134
C08108=1062.214,21.309,430.838,171.893,27.725,155.135
C08109=1062.219,21.558,430.823,171.895,27.727,155.135
C08110=1062.226,21.807,430.807,171.896,27.730,155.136
C08111=1062.231,22.057,430.792,171.898,27.733,155.136
C08112=1062.238,22.307,430.777,171.899,27.735,155.136
C08113=1062.244,22.556,430.761,171.900,27.738,155.137
C08114=1062.250,22.806,430.746,171.902,27.740,155.137
C08115=1062.256,23.054,430.730,171.903,27.743,155.137
C08116=1062.262,23.304,430.715,171.905,27.745,155.138
C08117=1062.268,23.554,430.699,171.906,27.748,155.138
C08118=1062.274,23.803,430.684,171.908,27.750,155.138
C08119=1062.280,24.053,430.668,171.909,27.753,155.139
C08120=1062.287,24.302,430.653,171.910,27.755,155.139
C08121=1062.292,24.552,430.637,171.912,27.758,155.139
C08122=1062.298,24.800,430.622,171.913,27.761,155.140
C08123=1062.304,25.050,430.606,171.915,27.763,155.140
C08124=1062.311,25.299,430.591,171.916,27.766,155.140
C08125=1062.316,25.549,430.575,171.918,27.768,155.141
C08126=1062.322,25.799,430.559,171.919,27.771,155.141
C08127=1062.329,26.048,430.544,171.921,27.773,155.141
C08128=1062.335,26.298,430.528,171.922,27.776,155.142
C08129=1062.341,26.547,430.513,171.923,27.778,155.142
C08130=1062.347,26.797,430.496,171.925,27.781,155.142
C08131=1062.353,27.046,430.481,171.926,27.783,155.143
C08132=1062.359,27.295,430.465,171.928,27.786,155.143
C08133=1062.365,27.545,430.451,171.930,27.789,155.143
C08134=1062.371,27.794,430.434,171.931,27.791,155.144
C08135=1062.377,28.044,430.419,171.933,27.794,155.144
C08136=1062.383,28.293,430.403,171.933,27.796,155.144
C08137=1062.389,28.542,430.387,171.935,27.798,155.145
C08138=1062.396,28.792,430.372,171.936,27.801,155.145
C08139=1062.402,29.041,430.356,171.938,27.804,155.145
C08140=1062.407,29.291,430.340,171.940,27.806,155.146
C08141=1062.413,29.541,430.324,171.941,27.809,155.146
C08142=1062.420,29.824,430.306,171.943,27.812,155.147
C08143=1062.427,30.109,430.288,171.944,27.815,155.147
C08144=1062.434,30.393,430.270,171.946,27.818,155.147
C08145=1062.441,30.678,430.253,171.947,27.820,155.148
C08146=1062.447,30.927,430.236,171.949,27.823,155.148
C08147=1062.453,31.176,430.220,171.950,27.825,155.148
C08148=1062.458,31.426,430.204,171.952,27.828,155.149
C08149=1062.465,31.675,430.189,171.953,27.831,155.149
C08150=1062.471,31.925,430.173,171.955,27.833,155.150
C08151=1062.477,32.174,430.156,171.956,27.836,155.150
C08152=1062.483,32.424,430.141,171.957,27.839,155.150
C08153=1062.489,32.673,430.125,171.959,27.841,155.151
C08154=1062.495,32.922,430.109,171.960,27.844,155.151
C08155=1062.501,33.172,430.093,171.962,27.846,155.151
C08156=1062.507,33.422,430.077,171.963,27.849,155.152
C08157=1062.514,33.671,430.061,171.965,27.852,155.152
C08158=1062.519,33.920,430.045,171.966,27.854,155.152
C08159=1062.525,34.169,430.029,171.967,27.857,155.153
C08160=1062.530,34.419,430.014,171.969,27.859,155.153
C08161=1062.536,34.668,429.997,171.970,27.862,155.153
C08162=1062.544,34.918,429.981,171.972,27.864,155.154
C08163=1062.550,35.167,429.965,171.973,27.867,155.154
C08164=1062.556,35.417,429.949,171.975,27.869,155.155
C08165=1062.561,35.666,429.933,171.976,27.872,155.155
C08166=1062.568,35.916,429.918,171.977,27.874,155.155
C08167=1062.574,36.165,429.901,171.979,27.877,155.156
C08168=1062.580,36.414,429.885,171.980,27.880,155.156
C08169=1062.586,36.664,429.869,171.982,27.882,155.156
C08170=1062.592,36.913,429.853,171.984,27.885,155.157
C08171=1062.598,37.163,429.838,171.985,27.888,155.157
C08172=1062.604,37.412,429.821,171.986,27.890,155.157
C08173=1062.610,37.661,429.805,171.987,27.893,155.158
C08174=1062.616,37.911,429.789,171.989,27.895,155.158
C08175=1062.622,38.160,429.773,171.990,27.898,155.158
C08176=1062.628,38.409,429.756,171.992,27.900,155.159
C08177=1062.634,38.659,429.740,171.994,27.903,155.159
C08178=1062.640,38.908,429.724,171.995,27.905,155.159
C08179=1062.646,39.157,429.708,171.996,27.908,155.160
C08180=1062.652,39.407,429.691,171.997,27.911,155.160
C08181=1062.657,39.657,429.676,171.999,27.914,155.161
C08182=1062.663,39.906,429.660,172.000,27.916,155.161
C08183=1062.669,40.155,429.643,172.002,27.919,155.161
C08184=1062.675,40.405,429.627,172.004,27.922,155.162
C08185=1062.681,40.654,429.611,172.005,27.924,155.162
C08186=1062.687,40.903,429.595,172.006,27.926,155.162
C08187=1062.694,41.153,429.578,172.007,27.929,155.163
C08188=1062.700,41.403,429.562,172.009,27.932,155.163
C08189=1062.706,41.652,429.545,172.011,27.934,155.164
C08190=1062.712,41.902,429.529,172.012,27.937,155.164
C08191=1062.717,42.151,429.513,172.014,27.940,155.164
C08192=1062.723,42.400,429.497,172.015,27.942,155.165
C08193=1062.730,42.649,429.480,172.016,27.945,155.165
C08194=1062.736,42.898,429.463,172.017,27.947,155.165
C08195=1062.742,43.148,429.447,172.019,27.950,155.166
C08196=1062.748,43.397,429.431,172.021,27.952,155.166
C08197=1062.753,43.646,429.415,172.022,27.955,155.166
C08198=1062.760,43.896,429.398,172.024,27.958,155.167
C08199=1062.766,44.146,429.382,172.025,27.961,155.167
C08200=1062.772,44.395,429.366,172.026,27.963,155.168
C08201=1062.777,44.645,429.349,172.027,27.966,155.168
C08202=1062.783,44.894,429.332,172.029,27.968,155.168
C08203=1062.789,45.143,429.316,172.031,27.971,155.169
C08204=1062.795,45.392,429.299,172.032,27.974,155.169
C08205=1062.801,45.642,429.282,172.034,27.977,155.170
C08206=1062.807,45.926,429.264,172.035,27.980,155.170
C08207=1062.814,46.211,429.245,172.037,27.983,155.170
C08208=1062.821,46.495,429.226,172.038,27.986,155.171
C08209=1062.827,46.779,429.208,172.040,27.989,155.171
C08210=1062.833,47.028,429.191,172.041,27.992,155.172
C08211=1062.839,47.277,429.174,172.043,27.994,155.172
C08212=1062.846,47.527,429.158,172.044,27.997,155.172
C08213=1062.851,47.777,429.141,172.045,27.999,155.173
C08214=1062.857,48.026,429.124,172.047,28.002,155.173
C08215=1062.863,48.275,429.108,172.048,28.005,155.174
C08216=1062.869,48.524,429.091,172.050,28.008,155.174
C08217=1062.874,48.774,429.074,172.051,28.010,155.174
C08218=1062.881,49.023,429.058,172.053,28.013,155.175
C08219=1062.887,49.272,429.041,172.054,28.015,155.175
C08220=1062.892,49.523,429.024,172.055,28.018,155.175
C08221=1062.898,49.772,429.008,172.057,28.021,155.176
C08222=1062.905,50.021,428.991,172.058,28.024,155.176
C08223=1062.911,50.270,428.975,172.060,28.026,155.176
C08224=1062.916,50.520,428.958,172.061,28.029,155.177
C08225=1062.922,50.768,428.941,172.063,28.031,155.177
C08226=1062.929,51.018,428.924,172.064,28.034,155.178
C08227=1062.935,51.268,428.908,172.065,28.037,155.178
C08228=1062.940,51.517,428.890,172.067,28.039,155.178
C08229=1062.946,51.766,428.874,172.068,28.042,155.179
C08230=1062.952,52.016,428.858,172.070,28.045,155.179
C08231=1062.958,52.265,428.840,172.071,28.047,155.180
C08232=1062.964,52.515,428.824,172.073,28.050,155.180
C08233=1062.970,52.764,428.807,172.074,28.052,155.180
C08234=1062.976,53.013,428.790,172.075,28.055,155.181
C08235=1062.982,53.263,428.773,172.077,28.058,155.181
C08236=1062.988,53.512,428.757,172.078,28.061,155.181
C08237=1062.994,53.761,428.740,172.080,28.063,155.182
C08238=1063.000,54.011,428.723,172.081,28.066,155.182
C08239=1063.006,54.260,428.706,172.083,28.068,155.182
C08240=1063.012,54.510,428.689,172.085,28.071,155.183
C08241=1063.018,54.759,428.672,172.085,28.074,155.183
C08242=1063.028,55.173,428.644,172.087,28.078,155.184
C08243=1063.038,55.588,428.616,172.091,28.082,155.184
C08244=1063.048,56.002,428.588,172.093,28.087,155.185
C08245=1063.058,56.416,428.560,172.095,28.091,155.186
C08246=1063.064,56.667,428.543,172.097,28.094,155.186
C08247=1063.070,56.916,428.526,172.098,28.096,155.186
C08248=1063.075,57.165,428.509,172.099,28.099,155.187
C08249=1063.082,57.414,428.492,172.101,28.102,155.187
C08250=1063.088,57.664,428.476,172.102,28.105,155.188
C08251=1063.094,57.913,428.458,172.104,28.107,155.188
C08252=1063.100,58.162,428.442,172.105,28.110,155.188
C08253=1063.107,58.412,428.425,172.107,28.112,155.189
C08254=1063.112,58.661,428.407,172.108,28.115,155.189
C08255=1063.118,58.910,428.391,172.109,28.117,155.189
C08256=1063.125,59.160,428.373,172.111,28.120,155.190
C08257=1063.130,59.409,428.357,172.112,28.123,155.190
C08258=1063.136,59.658,428.340,172.114,28.126,155.191
C08259=1063.143,59.908,428.323,172.116,28.128,155.191
C08260=1063.148,60.157,428.305,172.117,28.131,155.191
C08261=1063.155,60.406,428.288,172.119,28.133,155.192
C08262=1063.161,60.656,428.271,172.119,28.136,155.192
C08263=1063.167,60.905,428.254,172.121,28.138,155.192
C08264=1063.174,61.154,428.237,172.123,28.141,155.193
C08265=1063.179,61.404,428.220,172.124,28.144,155.193
C08266=1063.189,61.772,428.195,172.127,28.147,155.194
C08267=1063.198,62.140,428.169,172.128,28.151,155.194
C08268=1063.206,62.508,428.144,172.130,28.155,155.195
C08269=1063.215,62.877,428.119,172.133,28.159,155.195
C08270=1063.221,63.126,428.102,172.134,28.162,155.196
C08271=1063.228,63.375,428.084,172.136,28.164,155.196
C08272=1063.233,63.624,428.067,172.137,28.167,155.196
C08273=1063.240,63.874,428.050,172.138,28.169,155.197
C08274=1063.246,64.123,428.033,172.140,28.172,155.197
C08275=1063.252,64.373,428.015,172.141,28.174,155.198
C08276=1063.258,64.622,427.999,172.143,28.177,155.198
C08277=1063.264,64.871,427.982,172.144,28.180,155.198
C08278=1063.270,65.121,427.964,172.146,28.183,155.199
C08279=1063.276,65.370,427.947,172.148,28.186,155.199
C08280=1063.282,65.619,427.929,172.148,28.188,155.199
C08281=1063.287,65.869,427.912,172.150,28.190,155.200
C08282=1063.294,66.118,427.895,172.151,28.193,155.200
C08283=1063.300,66.368,427.877,172.153,28.196,155.201
C08284=1063.306,66.616,427.860,172.154,28.199,155.201
C08285=1063.312,66.866,427.842,172.156,28.202,155.201
C08286=1063.318,67.115,427.824,172.158,28.204,155.202
C08287=1063.324,67.364,427.808,172.159,28.207,155.202
C08288=1063.330,67.614,427.790,172.160,28.209,155.203
C08289=1063.335,67.863,427.773,172.161,28.212,155.203
C08290=1063.342,68.113,427.755,172.163,28.215,155.203
C08291=1063.348,68.362,427.738,172.165,28.217,155.204
C08292=1063.354,68.611,427.720,172.166,28.220,155.204
C08293=1063.359,68.860,427.702,172.168,28.223,155.204
C08294=1063.365,69.109,427.685,172.169,28.225,155.205
C08295=1063.371,69.360,427.668,172.170,28.228,155.205
C08296=1063.377,69.609,427.651,172.172,28.231,155.206
C08297=1063.384,69.858,427.633,172.173,28.233,155.206
C08298=1063.389,70.107,427.616,172.175,28.236,155.206
C08299=1063.395,70.357,427.598,172.176,28.238,155.207
C08300=1063.401,70.606,427.580,172.178,28.241,155.207
C08301=1063.407,70.856,427.562,172.180,28.244,155.207
C08302=1063.413,71.104,427.545,172.180,28.247,155.208
C08303=1063.419,71.353,427.528,172.182,28.249,155.208
C08304=1063.425,71.603,427.510,172.183,28.252,155.209
C08305=1063.430,71.852,427.492,172.185,28.255,155.209
C08306=1063.436,72.102,427.474,172.186,28.258,155.210
C08307=1063.443,72.351,427.457,172.188,28.260,155.210
C08308=1063.449,72.600,427.439,172.190,28.263,155.210
C08309=1063.454,72.849,427.422,172.191,28.265,155.211
C08310=1063.460,73.099,427.404,172.192,28.268,155.211
C08311=1063.466,73.348,427.386,172.193,28.271,155.211
C08312=1063.472,73.598,427.368,172.195,28.274,155.212
C08313=1063.478,73.847,427.351,172.197,28.276,155.212
C08314=1063.484,74.096,427.333,172.198,28.279,155.213
C08315=1063.490,74.345,427.315,172.200,28.281,155.213
C08316=1063.496,74.595,427.297,172.201,28.284,155.213
C08317=1063.502,74.844,427.280,172.203,28.287,155.214
C08318=1063.508,75.093,427.262,172.204,28.289,155.214
C08319=1063.514,75.342,427.244,172.205,28.292,155.215
C08320=1063.520,75.592,427.226,172.207,28.295,155.215
C08321=1063.526,75.841,427.209,172.208,28.298,155.215
C08322=1063.532,76.091,427.191,172.210,28.300,155.216
C08323=1063.538,76.340,427.174,172.212,28.303,155.216
C08324=1063.544,76.589,427.155,172.213,28.306,155.216
C08325=1063.550,76.838,427.137,172.215,28.308,155.217
C08326=1063.556,77.088,427.120,172.215,28.311,155.217
C08327=1063.562,77.337,427.102,172.217,28.314,155.218
C08328=1063.567,77.586,427.084,172.218,28.316,155.218
C08329=1063.574,77.835,427.065,172.220,28.319,155.218
C08330=1063.581,78.119,427.046,172.222,28.322,155.219
C08331=1063.587,78.403,427.025,172.223,28.325,155.219
C08332=1063.594,78.688,427.005,172.225,28.328,155.220
C08333=1063.601,78.971,426.984,172.227,28.331,155.220
C08334=1063.607,79.221,426.966,172.228,28.334,155.221
C08335=1063.612,79.470,426.949,172.229,28.337,155.221
C08336=1063.618,79.719,426.931,172.231,28.339,155.221
C08337=1063.624,79.968,426.912,172.233,28.342,155.222
C08338=1063.630,80.217,426.895,172.234,28.345,155.222
C08339=1063.636,80.467,426.877,172.236,28.348,155.223
C08340=1063.641,80.716,426.858,172.237,28.350,155.223
C08341=1063.648,80.966,426.840,172.239,28.353,155.223
C08342=1063.653,81.215,426.822,172.240,28.356,155.224
C08343=1063.659,81.465,426.804,172.241,28.359,155.224
C08344=1063.665,81.713,426.786,172.243,28.361,155.225
C08345=1063.671,81.963,426.768,172.244,28.364,155.225
C08346=1063.677,82.211,426.750,172.246,28.366,155.225
C08347=1063.683,82.461,426.732,172.248,28.369,155.226
C08348=1063.688,82.711,426.713,172.249,28.372,155.226
C08349=1063.694,82.959,426.695,172.251,28.375,155.226
C08350=1063.700,83.209,426.677,172.251,28.377,155.227
C08351=1063.706,83.458,426.660,172.253,28.380,155.227
C08352=1063.712,83.707,426.641,172.254,28.383,155.228
C08353=1063.719,83.957,426.623,172.256,28.385,155.228
C08354=1063.724,84.205,426.605,172.258,28.388,155.228
C08355=1063.730,84.455,426.587,172.259,28.391,155.229
C08356=1063.736,84.705,426.568,172.261,28.394,155.229
C08357=1063.742,84.954,426.550,172.262,28.396,155.230
C08358=1063.748,85.203,426.532,172.264,28.399,155.230
C08359=1063.754,85.452,426.514,172.265,28.401,155.230
C08360=1063.760,85.701,426.496,172.266,28.404,155.231
C08361=1063.766,85.951,426.477,172.268,28.407,155.231
C08362=1063.771,86.200,426.459,172.269,28.410,155.232
C08363=1063.777,86.449,426.440,172.271,28.412,155.232
C08364=1063.783,86.699,426.422,172.273,28.415,155.232
C08365=1063.789,86.947,426.404,172.274,28.418,155.233
C08366=1063.795,87.197,426.386,172.276,28.421,155.233
C08367=1063.802,87.446,426.368,172.277,28.423,155.233
C08368=1063.807,87.696,426.349,172.278,28.425,155.234
C08369=1063.813,87.945,426.331,172.280,28.428,155.234
C08370=1063.819,88.194,426.313,172.281,28.431,155.235
C08371=1063.826,88.443,426.294,172.283,28.434,155.235
C08372=1063.831,88.692,426.277,172.284,28.437,155.235
C08373=1063.837,88.942,426.257,172.286,28.439,155.236
C08374=1063.843,89.191,426.239,172.288,28.442,155.236
C08375=1063.849,89.441,426.221,172.289,28.444,155.237
C08376=1063.855,89.689,426.202,172.291,28.447,155.237
C08377=1063.861,89.939,426.185,172.292,28.450,155.237
C08378=1063.867,90.188,426.165,172.293,28.452,155.238
C08379=1063.872,90.437,426.148,172.295,28.455,155.238
C08380=1063.879,90.687,426.129,172.296,28.458,155.239
C08381=1063.885,90.936,426.110,172.298,28.461,155.239
C08382=1063.891,91.186,426.092,172.299,28.463,155.239
C08383=1063.897,91.434,426.074,172.301,28.466,155.240
C08384=1063.902,91.684,426.054,172.303,28.468,155.240
C08385=1063.908,91.933,426.036,172.304,28.471,155.240
C08386=1063.914,92.182,426.018,172.306,28.474,155.241
C08387=1063.920,92.431,425.999,172.307,28.477,155.241
C08388=1063.926,92.681,425.981,172.308,28.479,155.242
C08389=1063.932,92.930,425.962,172.310,28.482,155.242
C08390=1063.938,93.179,425.943,172.311,28.485,155.242
C08391=1063.943,93.428,425.924,172.313,28.488,155.243
C08392=1063.949,93.678,425.906,172.314,28.490,155.243
C08393=1063.954,93.927,425.887,172.316,28.493,155.244
C08394=1063.961,94.211,425.866,172.318,28.496,155.244
C08395=1063.968,94.495,425.845,172.319,28.499,155.245
C08396=1063.975,94.779,425.824,172.321,28.503,155.245
C08397=1063.982,95.062,425.802,172.323,28.506,155.246
C08398=1063.988,95.312,425.784,172.325,28.508,155.246
C08399=1063.993,95.561,425.765,172.325,28.511,155.246
C08400=1064.000,95.810,425.747,172.327,28.514,155.247
C08401=1064.005,96.059,425.727,172.329,28.516,155.247
C08402=1064.012,96.308,425.709,172.330,28.519,155.248
C08403=1064.017,96.558,425.690,172.332,28.522,155.248
C08404=1064.023,96.807,425.672,172.333,28.525,155.248
C08405=1064.029,97.056,425.653,172.335,28.527,155.249
C08406=1064.035,97.305,425.634,172.337,28.530,155.249
C08407=1064.041,97.555,425.615,172.338,28.532,155.249
C08408=1064.047,97.804,425.596,172.340,28.535,155.250
C08409=1064.052,98.053,425.577,172.342,28.538,155.250
C08410=1064.059,98.302,425.559,172.342,28.540,155.251
C08411=1064.065,98.552,425.541,172.344,28.543,155.251
C08412=1064.070,98.801,425.521,172.345,28.546,155.251
C08413=1064.077,99.050,425.503,172.347,28.549,155.252
C08414=1064.083,99.300,425.483,172.349,28.552,155.252
C08415=1064.089,99.549,425.465,172.350,28.554,155.253
C08416=1064.094,99.797,425.446,172.352,28.557,155.253
C08417=1064.100,100.046,425.427,172.353,28.559,155.253
C08418=1064.106,100.296,425.408,172.355,28.562,155.254
C08419=1064.113,100.545,425.389,172.357,28.565,155.254
C08420=1064.118,100.794,425.370,172.358,28.568,155.255
C08421=1064.124,101.044,425.351,172.360,28.570,155.255
C08422=1064.130,101.293,425.332,172.361,28.573,155.255
C08423=1064.135,101.542,425.313,172.362,28.576,155.256
C08424=1064.141,101.791,425.294,172.364,28.578,155.256
C08425=1064.148,102.040,425.275,172.365,28.581,155.257
C08426=1064.153,102.290,425.256,172.367,28.584,155.257
C08427=1064.159,102.539,425.237,172.368,28.587,155.257
C08428=1064.165,102.789,425.218,172.370,28.589,155.258
C08429=1064.170,103.037,425.199,172.372,28.592,155.258
C08430=1064.176,103.286,425.180,172.373,28.595,155.259
C08431=1064.182,103.536,425.161,172.375,28.598,155.259
C08432=1064.188,103.785,425.142,172.377,28.600,155.259
C08433=1064.194,104.034,425.123,172.378,28.603,155.260
C08434=1064.200,104.284,425.104,172.380,28.606,155.260
C08435=1064.206,104.533,425.084,172.381,28.609,155.261
C08436=1064.211,104.781,425.066,172.383,28.611,155.261
C08437=1064.217,105.031,425.046,172.384,28.614,155.261
C08438=1064.223,105.280,425.027,172.385,28.617,155.262
C08439=1064.229,105.529,425.008,172.387,28.619,155.262
C08440=1064.235,105.779,424.989,172.388,28.622,155.263
C08441=1064.241,106.028,424.970,172.390,28.625,155.263
C08442=1064.247,106.277,424.950,172.392,28.628,155.263
C08443=1064.252,106.526,424.931,172.393,28.631,155.264
C08444=1064.259,106.775,424.912,172.395,28.633,155.264
C08445=1064.264,107.025,424.893,172.396,28.635,155.265
C08446=1064.270,107.274,424.874,172.398,28.638,155.265
C08447=1064.276,107.523,424.854,172.400,28.641,155.265
C08448=1064.282,107.771,424.835,172.401,28.644,155.266
C08449=1064.288,108.021,424.816,172.403,28.646,155.266
C08450=1064.293,108.270,424.797,172.405,28.649,155.267
C08451=1064.299,108.520,424.778,172.406,28.652,155.267
C08452=1064.305,108.769,424.758,172.408,28.655,155.267
C08453=1064.311,109.018,424.739,172.409,28.657,155.268
C08454=1064.317,109.267,424.720,172.411,28.660,155.268
C08455=1064.323,109.516,424.700,172.412,28.663,155.269
C08456=1064.329,109.765,424.681,172.413,28.666,155.269
C08457=1064.334,110.015,424.661,172.415,28.668,155.269
C08458=1064.342,110.298,424.640,172.417,28.671,155.270
C08459=1064.349,110.583,424.618,172.419,28.675,155.270
C08460=1064.355,110.867,424.595,172.421,28.677,155.271
C08461=1064.362,111.150,424.573,172.422,28.680,155.271
C08462=1064.368,111.400,424.554,172.424,28.683,155.272
C08463=1064.374,111.648,424.534,172.425,28.686,155.272
C08464=1064.380,111.898,424.515,172.427,28.688,155.272
C08465=1064.385,112.147,424.496,172.429,28.691,155.273
C08466=1064.391,112.396,424.476,172.430,28.694,155.273
C08467=1064.397,112.645,424.457,172.432,28.697,155.274
C08468=1064.403,112.895,424.437,172.433,28.699,155.274
C08469=1064.409,113.144,424.418,172.435,28.702,155.274
C08470=1064.415,113.393,424.398,172.437,28.705,155.275
C08471=1064.421,113.642,424.378,172.438,28.708,155.275
C08472=1064.426,113.891,424.359,172.440,28.710,155.276
C08473=1064.432,114.140,424.339,172.441,28.713,155.276
C08474=1064.438,114.390,424.320,172.443,28.716,155.276
C08475=1064.444,114.638,424.300,172.445,28.719,155.277
C08476=1064.450,114.888,424.281,172.446,28.721,155.277
C08477=1064.455,115.137,424.261,172.448,28.724,155.278
C08478=1064.461,115.386,424.241,172.450,28.727,155.278
C08479=1064.466,115.636,424.222,172.451,28.730,155.278
C08480=1064.472,115.885,424.202,172.453,28.733,155.279
C08481=1064.478,116.133,424.182,172.454,28.736,155.279
C08482=1064.484,116.383,424.162,172.456,28.738,155.280
C08483=1064.490,116.632,424.143,172.458,28.741,155.280
C08484=1064.495,116.881,424.123,172.459,28.744,155.281
C08485=1064.501,117.130,424.103,172.460,28.746,155.281
C08486=1064.507,117.380,424.083,172.461,28.749,155.281
C08487=1064.513,117.629,424.064,172.463,28.752,155.282
C08488=1064.518,117.878,424.044,172.465,28.755,155.282
C08489=1064.524,118.127,424.024,172.466,28.757,155.283
C08490=1064.529,118.376,424.004,172.468,28.760,155.283
C08491=1064.535,118.625,423.985,172.470,28.763,155.283
C08492=1064.541,118.874,423.965,172.471,28.766,155.284
C08493=1064.547,119.123,423.945,172.473,28.768,155.284
C08494=1064.553,119.373,423.925,172.474,28.771,155.285
C08495=1064.559,119.622,423.904,172.476,28.774,155.285
C08496=1064.564,119.872,423.885,172.478,28.777,155.285
C08497=1064.570,120.120,423.865,172.479,28.779,155.286
C08498=1064.576,120.369,423.845,172.481,28.782,155.286
C08499=1064.582,120.619,423.826,172.482,28.785,155.287
C08500=1064.587,120.868,423.805,172.484,28.788,155.287
C08501=1064.593,121.117,423.786,172.486,28.790,155.287
C08502=1064.599,121.365,423.766,172.487,28.793,155.288
C08503=1064.605,121.615,423.746,172.489,28.796,155.288
C08504=1064.610,121.864,423.726,172.491,28.799,155.289
C08505=1064.617,122.114,423.705,172.492,28.801,155.289
C08506=1064.623,122.363,423.686,172.494,28.804,155.289
C08507=1064.628,122.612,423.666,172.495,28.807,155.290
C08508=1064.634,122.861,423.646,172.497,28.810,155.290
C08509=1064.640,123.110,423.626,172.499,28.812,155.291
C08510=1064.646,123.359,423.606,172.500,28.815,155.291
C08511=1064.651,123.608,423.587,172.502,28.818,155.291
C08512=1064.658,123.857,423.566,172.504,28.820,155.292
C08513=1064.663,124.107,423.546,172.505,28.823,155.292
C08514=1064.669,124.355,423.526,172.507,28.826,155.293
C08515=1064.675,124.604,423.506,172.508,28.829,155.293
C08516=1064.681,124.854,423.486,172.510,28.831,155.293
C08517=1064.686,125.103,423.466,172.512,28.834,155.294
C08518=1064.693,125.352,423.446,172.513,28.837,155.294
C08519=1064.699,125.601,423.426,172.515,28.840,155.295
C08520=1064.705,125.850,423.406,172.517,28.842,155.295
C08521=1064.710,126.099,423.385,172.518,28.845,155.296
C08522=1064.717,126.383,423.362,172.521,28.849,155.296
C08523=1064.724,126.667,423.340,172.522,28.851,155.296
C08524=1064.730,126.951,423.316,172.524,28.855,155.297
C08525=1064.737,127.235,423.294,172.526,28.858,155.297
C08526=1064.743,127.484,423.274,172.528,28.860,155.298
C08527=1064.749,127.732,423.254,172.530,28.863,155.298
C08528=1064.755,127.982,423.233,172.531,28.866,155.299
C08529=1064.761,128.231,423.213,172.533,28.869,155.299
C08530=1064.767,128.480,423.193,172.535,28.871,155.299
C08531=1064.772,128.729,423.172,172.536,28.874,155.300
C08532=1064.779,128.978,423.152,172.538,28.877,155.300
C08533=1064.785,129.227,423.132,172.539,28.880,155.301
C08534=1064.790,129.476,423.112,172.541,28.882,155.301
C08535=1064.797,129.726,423.091,172.543,28.884,155.301
C08536=1064.803,129.975,423.071,172.544,28.887,155.302
C08537=1064.809,130.224,423.051,172.546,28.890,155.302
C08538=1064.814,130.473,423.031,172.548,28.893,155.302
C08539=1064.820,130.722,423.011,172.549,28.895,155.303
C08540=1064.826,130.971,422.991,172.551,28.898,155.303
C08541=1064.832,131.220,422.970,172.553,28.901,155.304
C08542=1064.838,131.470,422.950,172.554,28.904,155.304
C08543=1064.844,131.718,422.930,172.556,28.906,155.304
C08544=1064.849,131.968,422.909,172.557,28.909,155.305
C08545=1064.856,132.217,422.889,172.559,28.912,155.305
C08546=1064.861,132.466,422.868,172.561,28.915,155.306
C08547=1064.867,132.715,422.848,172.562,28.917,155.306
C08548=1064.873,132.964,422.828,172.564,28.920,155.307
C08549=1064.879,133.213,422.806,172.567,28.923,155.307
C08550=1064.885,133.462,422.786,172.568,28.926,155.307
C08551=1064.890,133.711,422.766,172.570,28.928,155.308
C08552=1064.896,133.960,422.746,172.571,28.931,155.308
C08553=1064.902,134.210,422.725,172.573,28.934,155.309
C08554=1064.907,134.459,422.704,172.575,28.937,155.309
C08555=1064.913,134.707,422.684,172.576,28.939,155.309
C08556=1064.919,134.957,422.663,172.578,28.942,155.310
C08557=1064.925,135.206,422.643,172.580,28.945,155.310
C08558=1064.930,135.455,422.622,172.581,28.948,155.311
C08559=1064.937,135.705,422.602,172.583,28.950,155.311
C08560=1064.943,135.953,422.580,172.585,28.953,155.311
C08561=1064.948,136.202,422.560,172.586,28.956,155.312
C08562=1064.955,136.452,422.540,172.588,28.958,155.312
C08563=1064.960,136.701,422.519,172.589,28.961,155.313
C08564=1064.965,136.949,422.498,172.591,28.964,155.313
C08565=1064.972,137.199,422.477,172.594,28.967,155.313
C08566=1064.977,137.448,422.457,172.595,28.970,155.314
C08567=1064.983,137.696,422.436,172.597,28.972,155.314
C08568=1064.989,137.946,422.415,172.599,28.975,155.315
C08569=1064.995,138.195,422.395,172.600,28.978,155.315
C08570=1065.001,138.443,422.374,172.602,28.981,155.315
C08571=1065.007,138.693,422.353,172.603,28.984,155.316
C08572=1065.012,138.942,422.333,172.605,28.987,155.316
C08573=1065.019,139.191,422.312,172.607,28.989,155.317
C08574=1065.024,139.440,422.291,172.608,28.992,155.317
C08575=1065.029,139.689,422.270,172.610,28.995,155.318
C08576=1065.036,139.938,422.249,172.612,28.997,155.318
C08577=1065.042,140.187,422.229,172.613,29.000,155.318
C08578=1065.047,140.436,422.208,172.616,29.003,155.319
C08579=1065.053,140.686,422.187,172.618,29.006,155.319
C08580=1065.058,140.935,422.166,172.619,29.009,155.320
C08581=1065.065,141.184,422.145,172.621,29.011,155.320
C08582=1065.070,141.433,422.125,172.622,29.014,155.320
C08583=1065.076,141.681,422.103,172.624,29.017,155.321
C08584=1065.082,141.931,422.082,172.626,29.019,155.321
C08585=1065.087,142.180,422.061,172.627,29.022,155.322
C08586=1065.094,142.464,422.037,172.630,29.026,155.322
C08587=1065.100,142.747,422.013,172.631,29.029,155.323
C08588=1065.107,143.031,421.989,172.633,29.032,155.323
C08589=1065.114,143.315,421.966,172.636,29.035,155.324
C08590=1065.120,143.563,421.945,172.637,29.038,155.324
C08591=1065.125,143.812,421.924,172.639,29.041,155.324
C08592=1065.131,144.062,421.903,172.641,29.043,155.325
C08593=1065.137,144.311,421.882,172.642,29.046,155.325
C08594=1065.143,144.560,421.860,172.644,29.049,155.326
C08595=1065.148,144.809,421.840,172.646,29.052,155.326
C08596=1065.155,145.058,421.819,172.648,29.054,155.326
C08597=1065.160,145.307,421.798,172.650,29.057,155.327
C08598=1065.166,145.556,421.777,172.651,29.060,155.327
C08599=1065.172,145.805,421.755,172.653,29.063,155.328
C08600=1065.178,146.055,421.734,172.655,29.065,155.328
C08601=1065.183,146.303,421.713,172.656,29.068,155.328
C08602=1065.190,146.552,421.692,172.658,29.071,155.329
C08603=1065.195,146.802,421.671,172.660,29.074,155.329
C08604=1065.202,147.050,421.650,172.662,29.077,155.330
C08605=1065.207,147.300,421.629,172.664,29.080,155.330
C08606=1065.213,147.549,421.608,172.665,29.082,155.331
C08607=1065.219,147.797,421.586,172.667,29.085,155.331
C08608=1065.225,148.046,421.565,172.669,29.088,155.331
C08609=1065.230,148.296,421.544,172.670,29.091,155.332
C08610=1065.236,148.545,421.523,172.672,29.093,155.332
C08611=1065.242,148.793,421.501,172.674,29.096,155.333
C08612=1065.248,149.043,421.480,172.676,29.099,155.333
C08613=1065.253,149.292,421.459,172.678,29.102,155.333
C08614=1065.259,149.541,421.438,172.680,29.104,155.334
C08615=1065.265,149.789,421.416,172.681,29.107,155.334
C08616=1065.271,150.039,421.395,172.683,29.110,155.335
C08617=1065.276,150.288,421.374,172.684,29.113,155.335
C08618=1065.283,150.537,421.352,172.686,29.116,155.336
C08619=1065.288,150.785,421.331,172.689,29.119,155.336
C08620=1065.293,151.035,421.309,172.690,29.122,155.336
C08621=1065.299,151.283,421.288,172.692,29.124,155.337
C08622=1065.305,151.533,421.267,172.694,29.127,155.337
C08623=1065.310,151.782,421.245,172.695,29.130,155.338
C08624=1065.317,152.031,421.224,172.697,29.132,155.338
C08625=1065.322,152.279,421.203,172.699,29.136,155.338
C08626=1065.328,152.529,421.181,172.701,29.139,155.339
C08627=1065.335,152.778,421.159,172.703,29.141,155.339
C08628=1065.340,153.026,421.138,172.704,29.144,155.340
C08629=1065.345,153.277,421.117,172.706,29.147,155.340
C08630=1065.351,153.525,421.095,172.708,29.149,155.341
C08631=1065.357,153.774,421.074,172.709,29.152,155.341
C08632=1065.362,154.023,421.052,172.712,29.155,155.341
C08633=1065.369,154.272,421.031,172.714,29.158,155.342
C08634=1065.375,154.521,421.009,172.715,29.160,155.342
C08635=1065.380,154.770,420.988,172.717,29.164,155.343
C08636=1065.386,155.019,420.966,172.719,29.166,155.343
C08637=1065.392,155.268,420.944,172.720,29.169,155.343
C08638=1065.398,155.517,420.923,172.723,29.172,155.344
C08639=1065.404,155.766,420.901,172.725,29.175,155.344
C08640=1065.409,156.015,420.880,172.726,29.178,155.345
C08641=1065.415,156.264,420.858,172.728,29.180,155.345
C08642=1065.421,156.513,420.836,172.729,29.184,155.346
C08643=1065.426,156.762,420.815,172.732,29.186,155.346
C08644=1065.433,157.011,420.793,172.734,29.189,155.346
C08645=1065.437,157.260,420.771,172.735,29.192,155.347
C08646=1065.444,157.509,420.749,172.737,29.195,155.347
C08647=1065.450,157.758,420.728,172.739,29.197,155.348
C08648=1065.455,158.007,420.706,172.741,29.200,155.348
C08649=1065.461,158.256,420.684,172.743,29.203,155.348
C08650=1065.468,158.540,420.660,172.745,29.206,155.349
C08651=1065.473,158.823,420.635,172.747,29.210,155.349
C08652=1065.480,159.106,420.610,172.749,29.213,155.350
C08653=1065.487,159.390,420.585,172.751,29.216,155.350
C08654=1065.493,159.639,420.563,172.753,29.219,155.351
C08655=1065.498,159.888,420.542,172.755,29.222,155.351
C08656=1065.505,160.136,420.519,172.756,29.225,155.352
C08657=1065.510,160.386,420.497,172.759,29.227,155.352
C08658=1065.517,160.635,420.476,172.761,29.230,155.352
C08659=1065.522,160.883,420.454,172.762,29.233,155.353
C08660=1065.528,161.133,420.433,172.764,29.236,155.353
C08661=1065.534,161.381,420.410,172.765,29.238,155.354
C08662=1065.539,161.630,420.388,172.768,29.242,155.354
C08663=1065.545,161.880,420.366,172.770,29.245,155.355
C08664=1065.550,162.128,420.344,172.771,29.247,155.355
C08665=1065.556,162.377,420.321,172.773,29.250,155.356
C08666=1065.562,162.626,420.300,172.775,29.253,155.356
C08667=1065.566,162.875,420.278,172.777,29.256,155.356
C08668=1065.573,163.124,420.256,172.779,29.259,155.357
C08669=1065.578,163.373,420.233,172.781,29.262,155.357
C08670=1065.583,163.622,420.211,172.782,29.265,155.358
C08671=1065.590,163.871,420.189,172.785,29.268,155.358
C08672=1065.595,164.120,420.167,172.786,29.271,155.359
C08673=1065.600,164.369,420.145,172.788,29.274,155.359
C08674=1065.606,164.618,420.123,172.790,29.276,155.359
C08675=1065.612,164.867,420.100,172.791,29.280,155.360
C08676=1065.617,165.116,420.079,172.794,29.283,155.360
C08677=1065.623,165.365,420.056,172.796,29.285,155.361
C08678=1065.629,165.614,420.034,172.797,29.289,155.361
C08679=1065.634,165.862,420.011,172.799,29.291,155.362
C08680=1065.640,166.111,419.990,172.802,29.294,155.362
C08681=1065.646,166.360,419.967,172.803,29.297,155.363
C08682=1065.651,166.610,419.945,172.805,29.300,155.363
C08683=1065.657,166.858,419.923,172.806,29.303,155.363
C08684=1065.662,167.107,419.900,172.809,29.306,155.364
C08685=1065.668,167.357,419.878,172.811,29.309,155.364
C08686=1065.674,167.605,419.856,172.812,29.312,155.365
C08687=1065.679,167.854,419.834,172.814,29.314,155.365
C08688=1065.685,168.103,419.811,172.817,29.318,155.366
C08689=1065.691,168.352,419.789,172.818,29.321,155.366
C08690=1065.697,168.601,419.766,172.820,29.323,155.367
C08691=1065.702,168.849,419.744,172.822,29.326,155.367
C08692=1065.708,169.099,419.722,172.824,29.329,155.367
C08693=1065.714,169.348,419.699,172.826,29.332,155.368
C08694=1065.719,169.597,419.677,172.828,29.335,155.368
C08695=1065.725,169.846,419.654,172.829,29.338,155.369
C08696=1065.730,170.094,419.633,172.832,29.341,155.369
C08697=1065.736,170.343,419.610,172.833,29.344,155.370
C08698=1065.742,170.592,419.587,172.835,29.346,155.370
C08699=1065.748,170.841,419.565,172.838,29.350,155.371
C08700=1065.754,171.090,419.542,172.839,29.353,155.371
C08701=1065.759,171.339,419.520,172.841,29.355,155.371
C08702=1065.764,171.588,419.498,172.843,29.358,155.372
C08703=1065.771,171.837,419.475,172.845,29.361,155.372
C08704=1065.776,172.086,419.453,172.847,29.364,155.373
C08705=1065.782,172.335,419.430,172.849,29.367,155.373
C08706=1065.788,172.584,419.407,172.851,29.370,155.373
C08707=1065.794,172.833,419.385,172.853,29.373,155.374
C08708=1065.799,173.081,419.363,172.855,29.376,155.374
C08709=1065.805,173.330,419.340,172.856,29.378,155.375
C08710=1065.810,173.579,419.317,172.859,29.382,155.375
C08711=1065.817,173.828,419.295,172.860,29.385,155.376
C08712=1065.822,174.077,419.272,172.862,29.387,155.376
C08713=1065.828,174.326,419.249,172.865,29.390,155.377
C08714=1065.835,174.609,419.223,172.866,29.393,155.377
C08715=1065.842,174.893,419.199,172.869,29.397,155.378
C08716=1065.848,175.175,419.173,172.872,29.400,155.378
C08717=1065.854,175.458,419.147,172.873,29.404,155.379
C08718=1065.860,175.707,419.124,172.876,29.406,155.379
C08719=1065.866,175.956,419.101,172.877,29.409,155.379
C08720=1065.872,176.205,419.079,172.879,29.412,155.380
C08721=1065.878,176.454,419.056,172.882,29.415,155.380
C08722=1065.883,176.703,419.034,172.883,29.418,155.381
C08723=1065.889,176.952,419.011,172.885,29.421,155.381
C08724=1065.895,177.201,418.988,172.888,29.424,155.382
C08725=1065.901,177.449,418.965,172.889,29.427,155.382
C08726=1065.907,177.698,418.942,172.891,29.430,155.382
C08727=1065.913,177.947,418.919,172.894,29.432,155.383
C08728=1065.918,178.196,418.896,172.895,29.435,155.383
C08729=1065.924,178.446,418.874,172.897,29.438,155.384
C08730=1065.930,178.694,418.851,172.900,29.441,155.384
C08731=1065.936,178.943,418.829,172.901,29.444,155.385
C08732=1065.942,179.192,418.806,172.903,29.447,155.385
C08733=1065.947,179.441,418.783,172.906,29.450,155.386
C08734=1065.953,179.690,418.760,172.907,29.453,155.386
C08735=1065.959,179.939,418.737,172.909,29.455,155.386
C08736=1065.965,180.187,418.715,172.912,29.458,155.387
C08737=1065.971,180.436,418.692,172.913,29.462,155.387
C08738=1065.977,180.685,418.669,172.915,29.464,155.388
C08739=1065.983,180.934,418.646,172.917,29.467,155.388
C08740=1065.988,181.183,418.623,172.919,29.470,155.389
C08741=1065.994,181.432,418.600,172.922,29.473,155.389
C08742=1066.000,181.681,418.577,172.923,29.476,155.389
C08743=1066.007,181.930,418.554,172.925,29.479,155.390
C08744=1066.013,182.179,418.531,172.928,29.482,155.390
C08745=1066.019,182.427,418.508,172.929,29.485,155.391
C08746=1066.024,182.676,418.485,172.931,29.488,155.391
C08747=1066.030,182.925,418.462,172.934,29.490,155.392
C08748=1066.036,183.174,418.439,172.935,29.493,155.392
C08749=1066.042,183.423,418.416,172.938,29.496,155.392
C08750=1066.048,183.671,418.394,172.940,29.499,155.393
C08751=1066.054,183.920,418.371,172.941,29.502,155.393
C08752=1066.060,184.170,418.347,172.944,29.505,155.394
C08753=1066.066,184.418,418.324,172.946,29.507,155.394
C08754=1066.072,184.667,418.301,172.948,29.511,155.395
C08755=1066.078,184.916,418.278,172.950,29.514,155.395
C08756=1066.083,185.165,418.254,172.952,29.517,155.396
C08757=1066.088,185.414,418.231,172.954,29.520,155.396
C08758=1066.094,185.662,418.208,172.956,29.523,155.396
C08759=1066.099,185.911,418.184,172.958,29.526,155.397
C08760=1066.105,186.160,418.161,172.960,29.529,155.397
C08761=1066.111,186.409,418.138,172.962,29.532,155.398
C08762=1066.116,186.658,418.114,172.964,29.535,155.398
C08763=1066.122,186.907,418.091,172.966,29.538,155.399
C08764=1066.128,187.156,418.068,172.969,29.541,155.399
C08765=1066.133,187.404,418.044,172.970,29.544,155.400
C08766=1066.139,187.653,418.021,172.972,29.547,155.400
C08767=1066.144,187.902,417.998,172.975,29.550,155.401
C08768=1066.150,188.151,417.973,172.976,29.553,155.401
C08769=1066.156,188.400,417.950,172.979,29.556,155.402
C08770=1066.162,188.648,417.927,172.981,29.560,155.402
C08771=1066.167,188.898,417.903,172.982,29.563,155.403
C08772=1066.173,189.147,417.880,172.985,29.566,155.403
C08773=1066.179,189.395,417.857,172.986,29.569,155.404
C08774=1066.184,189.644,417.833,172.989,29.572,155.404
C08775=1066.190,189.892,417.809,172.991,29.575,155.404
C08776=1066.195,190.141,417.786,172.993,29.578,155.405
C08777=1066.201,190.390,417.762,172.995,29.581,155.405
C08778=1066.207,190.673,417.736,172.998,29.585,155.406
C08779=1066.214,190.956,417.709,173.000,29.588,155.406
C08780=1066.220,191.238,417.682,173.002,29.591,155.407
C08781=1066.227,191.521,417.655,173.004,29.595,155.407
C08782=1066.232,191.770,417.632,173.007,29.598,155.408
C08783=1066.238,192.018,417.608,173.009,29.601,155.408
C08784=1066.244,192.268,417.584,173.010,29.604,155.409
C08785=1066.250,192.516,417.561,173.013,29.607,155.409
C08786=1066.255,192.766,417.537,173.015,29.610,155.410
C08787=1066.261,193.014,417.513,173.017,29.613,155.410
C08788=1066.267,193.262,417.490,173.019,29.616,155.411
C08789=1066.273,193.512,417.466,173.022,29.619,155.411
C08790=1066.279,193.760,417.442,173.023,29.622,155.412
C08791=1066.284,194.009,417.419,173.026,29.625,155.412
C08792=1066.290,194.258,417.395,173.028,29.629,155.413
C08793=1066.296,194.507,417.371,173.030,29.631,155.413
C08794=1066.301,194.756,417.347,173.032,29.635,155.414
C08795=1066.307,195.004,417.324,173.035,29.638,155.414
C08796=1066.313,195.253,417.299,173.036,29.641,155.414
C08797=1066.319,195.502,417.276,173.038,29.644,155.415
C08798=1066.324,195.751,417.252,173.041,29.647,155.415
C08799=1066.330,195.999,417.228,173.042,29.650,155.416
C08800=1066.336,196.248,417.205,173.045,29.653,155.416
C08801=1066.342,196.497,417.181,173.046,29.656,155.417
C08802=1066.348,196.746,417.157,173.049,29.659,155.417
C08803=1066.353,196.994,417.133,173.051,29.662,155.418
C08804=1066.360,197.244,417.109,173.053,29.665,155.418
C08805=1066.365,197.492,417.085,173.055,29.668,155.419
C08806=1066.371,197.741,417.062,173.058,29.671,155.419
C08807=1066.377,197.990,417.037,173.059,29.674,155.420
C08808=1066.383,198.239,417.014,173.062,29.677,155.420
C08809=1066.388,198.488,416.990,173.064,29.681,155.421
C08810=1066.395,198.737,416.966,173.066,29.684,155.421
C08811=1066.400,198.985,416.941,173.069,29.687,155.421
C08812=1066.406,199.233,416.918,173.071,29.690,155.422
C08813=1066.412,199.483,416.893,173.073,29.693,155.422
C08814=1066.418,199.731,416.869,173.075,29.696,155.423
C08815=1066.423,199.980,416.846,173.078,29.699,155.423
C08816=1066.430,200.229,416.822,173.079,29.702,155.424
C08817=1066.435,200.478,416.798,173.082,29.705,155.424
C08818=1066.441,200.727,416.774,173.084,29.708,155.425
C08819=1066.447,200.975,416.749,173.086,29.711,155.425
C08820=1066.453,201.224,416.726,173.088,29.714,155.426
C08821=1066.459,201.473,416.701,173.090,29.718,155.426
C08822=1066.465,201.721,416.677,173.092,29.721,155.427
C08823=1066.471,201.970,416.653,173.095,29.724,155.427
C08824=1066.477,202.219,416.629,173.097,29.727,155.428
C08825=1066.482,202.467,416.605,173.099,29.730,155.428
C08826=1066.488,202.717,416.580,173.102,29.734,155.429
C08827=1066.493,202.965,416.556,173.103,29.736,155.429
C08828=1066.500,203.214,416.532,173.106,29.740,155.429
C08829=1066.505,203.463,416.508,173.108,29.743,155.430
C08830=1066.510,203.711,416.483,173.110,29.746,155.431
C08831=1066.516,203.961,416.459,173.112,29.749,155.431
C08832=1066.522,204.209,416.435,173.115,29.752,155.431
C08833=1066.528,204.458,416.411,173.116,29.756,155.432
C08834=1066.534,204.707,416.386,173.119,29.759,155.433
C08835=1066.539,204.955,416.362,173.122,29.762,155.433
C08836=1066.545,205.204,416.337,173.123,29.765,155.433
C08837=1066.551,205.452,416.313,173.126,29.768,155.434
C08838=1066.557,205.702,416.288,173.128,29.771,155.434
C08839=1066.562,205.950,416.264,173.130,29.775,155.435
C08840=1066.568,206.199,416.240,173.132,29.778,155.435
C08841=1066.573,206.448,416.215,173.134,29.781,155.436
C08842=1066.598,207.493,416.113,173.288,29.857,155.441
C08843=1066.604,207.711,416.090,173.289,29.861,155.441
C08844=1066.609,207.930,416.068,173.291,29.865,155.442
C08845=1066.614,208.149,416.046,173.293,29.868,155.442
C08846=1066.620,208.367,416.024,173.294,29.872,155.443
C08847=1066.625,208.586,416.002,173.296,29.876,155.444
C08848=1066.629,208.804,415.979,173.297,29.879,155.444
C08849=1066.635,209.023,415.957,173.299,29.883,155.445
C08850=1066.640,209.241,415.935,173.302,29.887,155.446
C08851=1066.646,209.490,415.909,173.303,29.890,155.446
C08852=1066.652,209.739,415.884,173.305,29.894,155.447
C08853=1066.658,209.987,415.859,173.307,29.899,155.448
C08854=1066.664,210.236,415.834,173.309,29.902,155.448
C08855=1066.670,210.484,415.808,173.312,29.907,155.449
C08856=1066.676,210.733,415.783,173.313,29.911,155.450
C08857=1066.682,210.982,415.757,173.315,29.914,155.450
C08858=1066.688,211.231,415.732,173.317,29.919,155.451
C08859=1066.694,211.479,415.707,173.319,29.923,155.452
C08860=1066.700,211.727,415.682,173.321,29.927,155.453
C08861=1066.705,211.976,415.656,173.323,29.931,155.453
C08862=1066.711,212.225,415.630,173.325,29.935,155.454
C08863=1066.718,212.474,415.605,173.327,29.939,155.455
C08864=1066.723,212.723,415.579,173.329,29.943,155.455
C08865=1066.729,212.971,415.554,173.331,29.947,155.456
C08866=1066.736,213.220,415.528,173.333,29.951,155.457
C08867=1066.741,213.469,415.502,173.336,29.956,155.458
C08868=1066.747,213.716,415.477,173.337,29.959,155.458
C08869=1066.753,213.965,415.451,173.339,29.964,155.459
C08870=1066.759,214.214,415.425,173.341,29.968,155.460
C08871=1066.765,214.463,415.400,173.343,29.972,155.460
C08872=1066.770,214.712,415.374,173.346,29.976,155.461
C08873=1066.777,214.960,415.349,173.347,29.980,155.462
C08874=1066.783,215.208,415.323,173.350,29.984,155.463
C08875=1066.788,215.457,415.297,173.351,29.988,155.463
C08876=1066.795,215.706,415.271,173.353,29.992,155.464
C08877=1066.800,215.955,415.246,173.356,29.996,155.465
C08878=1066.806,216.204,415.220,173.357,30.000,155.465
C08879=1066.813,216.452,415.194,173.360,30.004,155.466
C08880=1066.818,216.700,415.169,173.361,30.008,155.467
C08881=1066.824,216.949,415.143,173.364,30.013,155.467
C08882=1066.829,217.198,415.117,173.365,30.016,155.468
C08883=1066.836,217.446,415.091,173.368,30.020,155.469
C08884=1066.841,217.695,415.065,173.370,30.025,155.470
C08885=1066.848,217.943,415.040,173.372,30.029,155.470
C08886=1066.853,218.192,415.013,173.374,30.032,155.471
C08887=1066.860,218.440,414.988,173.375,30.037,155.472
C08888=1066.866,218.689,414.963,173.378,30.041,155.472
C08889=1066.872,218.937,414.936,173.380,30.044,155.473
C08890=1066.878,219.186,414.911,173.382,30.049,155.474
C08891=1066.883,219.435,414.885,173.384,30.053,155.474
C08892=1066.890,219.683,414.859,173.387,30.057,155.475
C08893=1066.895,219.932,414.833,173.388,30.061,155.476
C08894=1066.902,220.181,414.806,173.391,30.065,155.476
C08895=1066.908,220.430,414.780,173.392,30.069,155.477
C08896=1066.914,220.678,414.754,173.395,30.073,155.478
C08897=1066.920,220.927,414.728,173.397,30.077,155.479
C08898=1066.926,221.176,414.703,173.399,30.081,155.479
C08899=1066.931,221.396,414.679,173.401,30.084,155.480
C08900=1066.937,221.617,414.656,173.402,30.088,155.480
C08901=1066.941,221.838,414.634,173.404,30.091,155.481
C08902=1066.947,222.058,414.610,173.407,30.095,155.482
C08903=1066.952,222.279,414.586,173.408,30.099,155.482
C08904=1066.957,222.500,414.564,173.410,30.102,155.483
C08905=1066.963,222.721,414.540,173.412,30.106,155.484
C08906=1066.968,222.942,414.516,173.413,30.110,155.484
C08907=1066.974,223.191,414.491,173.416,30.114,155.485
C08908=1066.980,223.439,414.464,173.418,30.117,155.486
C08909=1066.985,223.688,414.438,173.420,30.122,155.486
C08910=1066.992,223.936,414.412,173.422,30.126,155.487
C08911=1066.998,224.185,414.386,173.424,30.130,155.488
C08912=1067.003,224.434,414.360,173.426,30.134,155.488
C08913=1067.009,224.682,414.333,173.429,30.138,155.489
C08914=1067.015,224.930,414.307,173.430,30.142,155.490
C08915=1067.021,225.179,414.281,173.433,30.146,155.490
C08916=1067.027,225.428,414.254,173.435,30.150,155.491
C08917=1067.033,225.676,414.227,173.437,30.154,155.492
C08918=1067.039,225.925,414.202,173.440,30.158,155.493
C08919=1067.045,226.173,414.175,173.441,30.162,155.493
C08920=1067.051,226.422,414.149,173.444,30.166,155.494
C08921=1067.056,226.670,414.122,173.446,30.170,155.495
C08922=1067.063,226.919,414.097,173.448,30.174,155.495
C08923=1067.069,227.168,414.070,173.450,30.178,155.496
C08924=1067.075,227.416,414.043,173.452,30.182,155.497
C08925=1067.081,227.665,414.016,173.454,30.186,155.497
C08926=1067.087,227.913,413.991,173.457,30.190,155.498
C08927=1067.093,228.162,413.964,173.458,30.194,155.499
C08928=1067.099,228.411,413.937,173.461,30.198,155.499
C08929=1067.105,228.659,413.911,173.463,30.202,155.500
C08930=1067.111,228.907,413.885,173.465,30.206,155.501
C08931=1067.117,229.155,413.858,173.468,30.210,155.501
C08932=1067.122,229.404,413.832,173.469,30.214,155.502
C08933=1067.129,229.653,413.805,173.472,30.218,155.503
C08934=1067.135,229.902,413.779,173.474,30.222,155.503
C08935=1067.140,230.150,413.752,173.476,30.226,155.504
C08936=1067.146,230.399,413.725,173.478,30.230,155.505
C08937=1067.153,230.648,413.698,173.481,30.234,155.506
C08938=1067.158,230.896,413.672,173.482,30.238,155.506
C08939=1067.164,231.144,413.645,173.485,30.242,155.507
C08940=1067.170,231.393,413.618,173.487,30.246,155.508
C08941=1067.176,231.641,413.592,173.489,30.250,155.508
C08942=1067.182,231.890,413.565,173.492,30.254,155.509
C08943=1067.188,232.138,413.538,173.493,30.258,155.510
C08944=1067.194,232.387,413.511,173.496,30.262,155.510
C08945=1067.199,232.635,413.485,173.498,30.266,155.511
C08946=1067.206,232.884,413.458,173.500,30.270,155.512
C08947=1067.212,233.133,413.431,173.502,30.274,155.512
C08948=1067.217,233.381,413.404,173.505,30.278,155.513
C08949=1067.224,233.630,413.377,173.507,30.282,155.514
C08950=1067.230,233.878,413.350,173.509,30.286,155.515
C08951=1067.236,234.126,413.323,173.511,30.290,155.515
C08952=1067.241,234.374,413.297,173.513,30.294,155.516
C08953=1067.248,234.624,413.270,173.516,30.298,155.517
C08954=1067.253,234.872,413.243,173.518,30.302,155.517
C08955=1067.258,235.088,413.219,173.520,30.305,155.518
C08956=1067.263,235.306,413.195,173.522,30.309,155.519
C08957=1067.269,235.522,413.173,173.523,30.312,155.519
C08958=1067.274,235.739,413.148,173.526,30.316,155.520
C08959=1067.279,235.956,413.125,173.528,30.319,155.520
C08960=1067.284,236.172,413.101,173.529,30.323,155.521
C08961=1067.289,236.389,413.078,173.531,30.326,155.522
C08962=1067.295,236.606,413.055,173.534,30.330,155.522
C08963=1067.301,236.855,413.027,173.535,30.334,155.523
C08964=1067.306,237.103,413.000,173.538,30.338,155.524
C08965=1067.312,237.352,412.973,173.541,30.342,155.524
C08966=1067.319,237.600,412.946,173.542,30.346,155.525
C08967=1067.325,237.848,412.919,173.545,30.350,155.526
C08968=1067.331,238.098,412.892,173.547,30.353,155.526
C08969=1067.336,238.346,412.864,173.549,30.358,155.527
C08970=1067.342,238.594,412.837,173.552,30.362,155.528
C08971=1067.348,238.843,412.810,173.554,30.366,155.528
C08972=1067.355,239.091,412.783,173.556,30.369,155.529
C08973=1067.361,239.340,412.756,173.558,30.374,155.530
C08974=1067.366,239.588,412.729,173.561,30.378,155.530
C08975=1067.372,239.836,412.701,173.563,30.382,155.531
C08976=1067.378,240.085,412.674,173.565,30.385,155.532
C08977=1067.384,240.333,412.647,173.568,30.390,155.533
C08978=1067.391,240.582,412.620,173.570,30.394,155.533
C08979=1067.396,240.830,412.592,173.572,30.397,155.534
C08980=1067.402,241.078,412.565,173.575,30.401,155.535
C08981=1067.409,241.327,412.538,173.577,30.406,155.535
C08982=1067.414,241.576,412.510,173.579,30.409,155.536
C08983=1067.420,241.824,412.483,173.581,30.413,155.537
C08984=1067.426,242.072,412.456,173.584,30.417,155.537
C08985=1067.433,242.321,412.428,173.586,30.421,155.538
C08986=1067.438,242.569,412.401,173.588,30.425,155.539
C08987=1067.445,242.818,412.373,173.590,30.429,155.539
C08988=1067.450,243.067,412.346,173.593,30.433,155.540
C08989=1067.456,243.315,412.318,173.595,30.437,155.541
C08990=1067.462,243.563,412.291,173.597,30.441,155.541
C08991=1067.468,243.812,412.263,173.600,30.445,155.542
C08992=1067.474,244.060,412.236,173.602,30.449,155.543
C08993=1067.479,244.308,412.208,173.604,30.453,155.544
C08994=1067.486,244.557,412.181,173.607,30.457,155.544
C08995=1067.491,244.805,412.153,173.609,30.461,155.545
C08996=1067.498,245.054,412.125,173.611,30.465,155.546
C08997=1067.503,245.302,412.098,173.614,30.469,155.546
C08998=1067.509,245.551,412.070,173.616,30.473,155.547
C08999=1067.515,245.799,412.042,173.618,30.477,155.548
C09000=1067.522,246.047,412.015,173.621,30.481,155.548
C09001=1067.527,246.296,411.987,173.623,30.485,155.549
C09002=1067.533,246.544,411.960,173.626,30.489,155.550
C09003=1067.539,246.793,411.931,173.628,30.493,155.550
C09004=1067.545,247.041,411.903,173.630,30.497,155.551
C09005=1067.551,247.289,411.876,173.633,30.501,155.552
C09006=1067.556,247.538,411.848,173.635,30.505,155.553
C09007=1067.562,247.786,411.820,173.637,30.510,155.553
C09008=1067.568,248.035,411.793,173.640,30.513,155.554
C09009=1067.574,248.283,411.765,173.642,30.517,155.555
C09010=1067.580,248.531,411.736,173.644,30.522,155.555
C09011=1067.585,248.745,411.712,173.646,30.525,155.556
C09012=1067.590,248.959,411.689,173.649,30.529,155.557
C09013=1067.595,249.173,411.664,173.650,30.532,155.557
C09014=1067.600,249.385,411.640,173.652,30.535,155.558
C09015=1067.604,249.600,411.617,173.655,30.539,155.558
C09016=1067.610,249.813,411.593,173.656,30.542,155.559
C09017=1067.615,250.027,411.568,173.658,30.546,155.560
C09018=1067.620,250.240,411.544,173.661,30.549,155.560
C09019=1067.626,250.489,411.516,173.663,30.553,155.561
C09020=1067.631,250.737,411.488,173.665,30.557,155.562
C09021=1067.638,250.985,411.460,173.668,30.561,155.562
C09022=1067.643,251.233,411.432,173.670,30.565,155.563
C09023=1067.649,251.482,411.404,173.672,30.569,155.564
C09024=1067.655,251.731,411.375,173.675,30.573,155.564
C09025=1067.661,251.979,411.348,173.678,30.577,155.565
C09026=1067.667,252.227,411.320,173.679,30.581,155.566
C09027=1067.673,252.475,411.292,173.682,30.585,155.566
C09028=1067.679,252.724,411.263,173.685,30.589,155.567
C09029=1067.685,252.973,411.236,173.687,30.593,155.568
C09030=1067.691,253.221,411.208,173.689,30.597,155.569
C09031=1067.697,253.469,411.179,173.692,30.601,155.569
C09032=1067.703,253.718,411.150,173.694,30.605,155.570
C09033=1067.708,253.966,411.122,173.697,30.609,155.571
C09034=1067.715,254.214,411.095,173.699,30.613,155.571
C09035=1067.721,254.463,411.066,173.701,30.617,155.572
C09036=1067.726,254.710,411.038,173.704,30.621,155.573
C09037=1067.732,254.959,411.009,173.707,30.625,155.573
C09038=1067.738,255.208,410.981,173.708,30.629,155.574
C09039=1067.745,255.456,410.953,173.711,30.633,155.575
C09040=1067.751,255.704,410.925,173.714,30.637,155.575
C09041=1067.757,255.952,410.896,173.716,30.641,155.576
C09042=1067.763,256.201,410.868,173.718,30.645,155.577
C09043=1067.768,256.449,410.839,173.721,30.649,155.578
C09044=1067.775,256.697,410.812,173.723,30.653,155.578
C09045=1067.781,256.946,410.783,173.726,30.656,155.579
C09046=1067.787,257.194,410.754,173.728,30.661,155.580
C09047=1067.793,257.443,410.726,173.730,30.665,155.580
C09048=1067.798,257.691,410.698,173.733,30.668,155.581
C09049=1067.805,257.939,410.669,173.736,30.672,155.582
C09050=1067.811,258.187,410.641,173.739,30.677,155.582
C09051=1067.817,258.436,410.613,173.740,30.680,155.583
C09052=1067.823,258.683,410.584,173.743,30.684,155.584
C09053=1067.829,258.932,410.556,173.746,30.688,155.584
C09054=1067.835,259.180,410.527,173.748,30.692,155.585
C09055=1067.841,259.429,410.498,173.751,30.696,155.586
C09056=1067.847,259.677,410.469,173.753,30.700,155.586
C09057=1067.853,259.926,410.441,173.755,30.704,155.587
C09058=1067.860,260.173,410.413,173.758,30.708,155.588
C09059=1067.866,260.422,410.385,173.761,30.712,155.589
C09060=1067.872,260.670,410.356,173.763,30.716,155.589
C09061=1067.878,260.919,410.327,173.765,30.720,155.590
C09062=1067.884,261.167,410.298,173.768,30.724,155.591
C09063=1067.890,261.416,410.270,173.771,30.728,155.591
C09064=1067.896,261.664,410.241,173.773,30.732,155.592
C09065=1067.902,261.912,410.212,173.776,30.736,155.593
C09066=1067.908,262.161,410.184,173.779,30.739,155.593
C09067=1067.914,262.372,410.160,173.780,30.743,155.594
C09068=1067.919,262.585,410.135,173.782,30.746,155.595
C09069=1067.924,262.798,410.110,173.785,30.750,155.595
C09070=1067.929,263.010,410.085,173.787,30.753,155.596
C09071=1067.935,263.223,410.060,173.789,30.757,155.596
C09072=1067.941,263.434,410.036,173.791,30.760,155.597
C09073=1067.945,263.647,410.012,173.794,30.763,155.597
C09074=1067.951,263.860,409.987,173.796,30.767,155.598
C09075=1067.956,264.109,409.958,173.798,30.770,155.599
C09076=1067.962,264.356,409.929,173.801,30.774,155.599
C09077=1067.968,264.604,409.900,173.804,30.779,155.600
C09078=1067.974,264.852,409.871,173.805,30.782,155.601
C09079=1067.980,265.101,409.843,173.808,30.786,155.601
C09080=1067.986,265.349,409.813,173.811,30.791,155.602
C09081=1067.992,265.598,409.784,173.813,30.794,155.603
C09082=1067.998,265.846,409.755,173.816,30.798,155.604
C09083=1068.005,266.094,409.726,173.819,30.803,155.604
C09084=1068.010,266.342,409.696,173.821,30.806,155.605
C09085=1068.016,266.591,409.668,173.823,30.811,155.606
C09086=1068.022,266.838,409.639,173.826,30.815,155.606
C09087=1068.028,267.087,409.610,173.829,30.818,155.607
C09088=1068.033,267.335,409.581,173.831,30.823,155.608
C09089=1068.040,267.583,409.551,173.834,30.827,155.609
C09090=1068.046,267.831,409.522,173.837,30.831,155.609
C09091=1068.052,268.079,409.493,173.838,30.835,155.610
C09092=1068.058,268.328,409.464,173.841,30.839,155.611
C09093=1068.064,268.576,409.435,173.844,30.842,155.611
C09094=1068.070,268.824,409.406,173.847,30.846,155.612
C09095=1068.076,269.072,409.377,173.849,30.851,155.613
C09096=1068.082,269.321,409.347,173.852,30.854,155.613
C09097=1068.088,269.569,409.318,173.855,30.859,155.614
C09098=1068.094,269.817,409.288,173.857,30.863,155.615
C09099=1068.100,270.065,409.259,173.860,30.867,155.616
C09100=1068.106,270.314,409.230,173.862,30.871,155.616
C09101=1068.112,270.562,409.201,173.864,30.875,155.617
C09102=1068.118,270.810,409.171,173.867,30.878,155.618
C09103=1068.124,271.058,409.141,173.870,30.883,155.618
C09104=1068.130,271.306,409.112,173.873,30.887,155.619
C09105=1068.136,271.554,409.083,173.875,30.891,155.620
